Universal Robots URScript: MM_SIF408_Camera.script

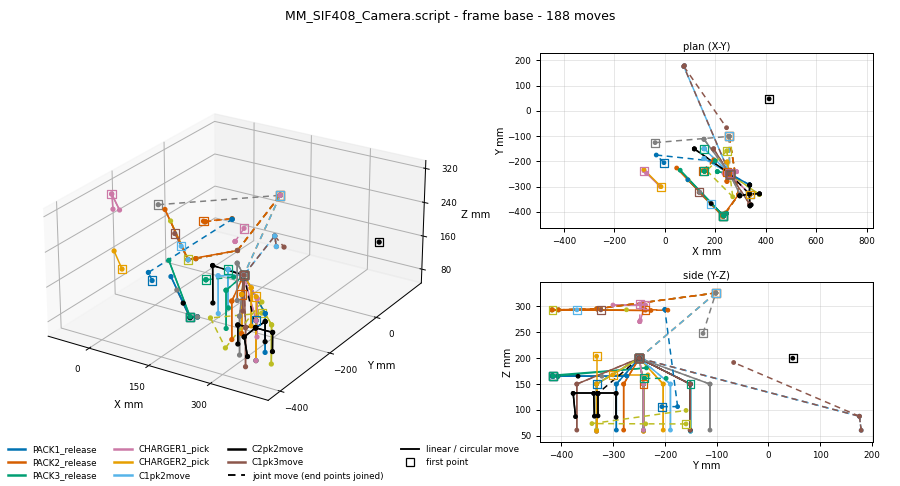
[picture p0: tool path of MM_SIF408_Camera.script in frame base, 188 of 288 moves have a stored position in this frame; points joined in program order, loops and branches not executed]
def MM_SIF408_Camera():
  global _hidden_verificationVariable=0
  step_count_84a8275e_68ac_46b0_8c6d_5b8d50443a58 = 0.0
  thread Step_Counter_Thread_a542c264_a21e_4968_aa71_40a8ac97ed48():
    while (True):
      step_count_84a8275e_68ac_46b0_8c6d_5b8d50443a58 = step_count_84a8275e_68ac_46b0_8c6d_5b8d50443a58 + 1.0
      sync()
    end
  end
  run Step_Counter_Thread_a542c264_a21e_4968_aa71_40a8ac97ed48()
  set_standard_analog_input_domain(0, 1)
  set_standard_analog_input_domain(1, 1)
  set_tool_analog_input_domain(0, 1)
  set_tool_analog_input_domain(1, 1)
  set_analog_outputdomain(0, 0)
  set_analog_outputdomain(1, 0)
  set_input_actions_to_default()
  modbus_add_signal("130.130.130.202", 255, 128, 2, "mm_insp_id", False)
  modbus_set_signal_update_frequency("mm_insp_id", 10)
  modbus_add_signal("130.130.130.202", 255, 129, 2, "mm_pht_stp_done", False)
  modbus_set_signal_update_frequency("mm_pht_stp_done", 10)
  modbus_add_signal("130.130.130.202", 255, 130, 2, "mm_res_ver", False)
  modbus_set_signal_update_frequency("mm_res_ver", 10)
  modbus_add_signal("130.130.130.202", 255, 131, 2, "c1_recorrect", False)
  modbus_set_signal_update_frequency("c1_recorrect", 10)
  modbus_add_signal("130.130.130.202", 255, 132, 2, "c2_recorrect", False)
  modbus_set_signal_update_frequency("c2_recorrect", 10)
  modbus_add_signal("130.130.130.202", 255, 133, 2, "c3_reconnect", False)
  modbus_set_signal_update_frequency("c3_reconnect", 10)
  modbus_add_signal("130.130.130.202", 255, 134, 2, "c4_reconnect", False)
  modbus_set_signal_update_frequency("c4_reconnect", 10)
  modbus_add_signal("130.130.130.202", 255, 135, 3, "mm_recv_inst", False)
  modbus_set_signal_update_frequency("mm_recv_inst", 10)
  modbus_add_signal("130.130.130.202", 255, 136, 3, "mm_pht_rdy_stp", False)
  modbus_set_signal_update_frequency("mm_pht_rdy_stp", 10)
  modbus_set_runstate_dependent_choice("mm_recv_inst",0)
  modbus_set_runstate_dependent_choice("mm_pht_rdy_stp",0)
  set_safety_mode_transition_hardness(1)
  set_tool_communication(True, 19200, 0, 1, 3.5, 3.5)
  set_tool_output_mode(1)
  set_tool_digital_output_mode(0, 1)
  set_tool_digital_output_mode(1, 1)
  set_tool_voltage(24)
  rtde_set_watchdog("speed_slider_mask", 10.0, "pause")
  rtde_set_watchdog("input_bit_registers0_to_31", 10.0, "pause")
  rtde_set_watchdog("input_bit_registers32_to_63", 10.0, "pause")
  set_tcp(p[0.0,0.0,0.105,0.0,0.0,0.0])
  set_gravity([0.0, 0.0, 9.82])
  set_target_payload(0.750000, [0.000000, 0.000000, 0.000000], [0.000000, 0.000000, 0.000000, 0.000000, 0.000000, 0.000000])
  global Plane_1_Pack=p[0.24802604835791223,-0.16109825037384065,0.07343232674968579,1.5770610514332666E-4,-1.6911666992609967E-4,-2.356123162082294]
  global Plane_2_Charger=p[-0.020825889928195812,-0.20923497632823723,0.10484675194267869,0.7321684888960871,-1.7600381110435173,-1.7743768301112888]
  global Plane_3_C1move=p[0.13168317783925995,-0.24026381339900515,0.1798744586307036,-1.7458660631601477,-0.7339675944130294,-1.7576520505834232]
  global abajo=p[0.236823956197105,-0.3085340218782548,0.07438383757948624,1.59760453662429E-5,-1.9018418942279844E-5,0.7930744342156013]
  global ChargerSafe_p=p[-.038219888098, -.126109356632, .247864627735, .768372410548, 1.381786852190, .427050797557]
  global ChargerSafe_q=[-2.290328532835165, -1.588600530279578, -1.8552938851973906, 3.426818033809969, -3.618186683716541, 5.475553405421589]
  global UL_HomePos_p=p[.254854540361, -.101396521086, .326005914920, .372294290291, 1.604272927406, .848817535244]
  global UL_HomePos_q=[-0.4437336060017767, -1.2677181226029575, -1.7403695179117786, 2.998681575604259, -2.3285643390928694, 5.484779635767351]
  global HomePos_p=p[.155172845975, -.134373233263, .327052937324, .372294290291, 1.604272927406, .848817535244]
  global HomePos_q=[-0.4437336060017767, -1.2677181226029575, -1.7403695179117786, 2.998681575604259, -2.3285643390928694, 5.484779635767351]
  global Waypoint_7_p=p[.235254426101, -.248279333010, .270600000000, -2.208471707321, 2.232557069129, -.003211421070]
  global Waypoint_7_q=[-0.4211163855529749, -1.695971462694982, -1.0919650932703284, 4.362995611362158, -4.714225695778342, 5.8733503607511075]
  global pl1_PK1up_2_p=p[.337707127627, -.331640151444, .150000000000, 2.209085410286, -2.230597199976, -.000628263705]
  global pl1_PK1up_2_q=[-0.4955539304835268, -2.270575736419687, -0.8287766003440309, 4.671022250611815, -4.717607275805612, 5.796412978798368]
  global pl1_PK1_1_p=p[.337708753286, -.331636321686, .059000000000, -2.208471682409, 2.232557092114, -.003211423953]
  global pl1_PK1_1_q=[-0.4967761842328837, -2.335801782331149, -1.1486863800200018, 5.0595087773604295, -4.714537561241828, 5.795733238729151]
  global pl1_PK1up_3_p=p[.337708753384, -.331636321739, .150000000045, -2.208471682402, 2.232557092122, -.003211423956]
  global pl1_PK1up_3_q=[-0.49668749848969007, -2.2676720609196863, -0.8351585073611147, 4.677851316512167, -4.714970187304847, 5.796430139558901]
  global Pack_aprox_1_p=p[.337708753236, -.331636321646, .203842313590, -2.208471707275, 2.232557069151, -.003211421080]
  global Pack_aprox_1_q=[-0.496372010829246, -2.3390319457501776, -0.44938640702618393, 4.363438999629054, -4.7153696447693765, 5.797111330864401]
  global pl1_PK2up_2_p=p[.246731843456, -.241011109916, .150000000097, 2.216981679034, -2.216426599865, .020673083567]
  global pl1_PK2up_2_q=[-0.3786656314116641, -1.6678189422546685, -1.7017298433113472, 4.951739825014103, -4.725262422761782, 5.9037751461208146]
  global p1_PK2_1_p=p[.246740908824, -.241008821032, .059000000000, 2.216983575726, -2.216446161785, .020720900301]
  global p1_PK2_1_q=[-0.3783922270214717, -1.8357706067986292, -1.9724640638814472, 5.390461636587837, -4.7249178522998685, 5.903567044989178]
  global pl1_PK2up_3_p=p[.246731843456, -.241011109916, .150000000097, 2.216981679034, -2.216426599865, .020673083567]
  global pl1_PK2up_3_q=[-0.3786656314116641, -1.6678189422546685, -1.7017298433113472, 4.951739825014103, -4.725262422761782, 5.9037751461208146]
  global Pack_aprox_3_p=p[.256529190168, -.247747736730, .304914735485, 2.216953502726, -2.216313122856, .021013179600]
  global Pack_aprox_3_q=[-0.45002005833990744, -1.7307120515452397, -1.4394096347220158, 4.751286312039589, -4.721256037152659, 5.839676484550372]
  global pl1_PK3up_2_p=p[.155982981866, -.150235111585, .149999999926, 2.204929412033, -2.228375225269, .020999038139]
  global pl1_PK3up_2_q=[-0.10405906347300053, -1.0147413698994976, -2.1858064021499084, 4.779384433270495, -4.726165068369075, 6.189377387251229]
  global pl1_PK3_1_p=p[.155974863337, -.150228231486, .059000001039, 2.204948002857, -2.228371305887, .020942580810]
  global pl1_PK3_1_q=[-0.10298431003644293, -1.1927496937335196, -2.5640957297909734, 5.335649879847573, -4.725692754745326, 6.190048722360077]
  global pl1_PK3up_3_p=p[.155982981866, -.150235111585, .149999999926, 2.204929412033, -2.228375225269, .020999038139]
  global pl1_PK3up_3_q=[-0.10405906347300053, -1.0147413698994976, -2.1858064021499084, 4.779384433270495, -4.726165068369075, 6.189377387251229]
  global C1_aprox1_p=p[-.133997460325, -.084557413006, .272269436052, .701218117570, 1.477825459734, .526200205067]
  global C1_aprox1_q=[-2.2378674310252507, -1.4936566577695842, -1.8069725022863468, 3.3775135356243458, -3.7069992982634132, 5.561485476738353]
  global C1_aprox2_p=p[-.161176845609, -.139586814883, .246569453044, 1.098520360937, 1.128202257975, .008787883398]
  global C1_aprox2_q=[-2.290389491672745, -1.5926356378882414, -1.8508182165530052, 3.416578818412902, -3.08727806453735, 5.46338959297019]
  global pl2_C1out_p=p[-.081795651010, -.237359145335, .302681515088, 1.127755706772, 1.089516743668, .021133838194]
  global pl2_C1out_q=[-2.1527147663452713, -1.5258578937050737, -1.651927109692683, 3.1816164398943436, -2.933001372406314, 5.5322042515010725]
  global pl2_C1_p=p[-.017768025182, -.300045052232, .302675455173, 1.127760213979, 1.089524808365, .021174235875]
  global pl2_C1_q=[-1.7215911662326384, -1.440872933618568, -1.7285842813986232, 3.1710747540129964, -2.5018731616546397, 5.52987656907406]
  global pl2_C1out_1_p=p[-.081795651010, -.237359145335, .302681515088, 1.127755706772, 1.089516743668, .021133838194]
  global pl2_C1out_1_q=[-2.1527147663452713, -1.5258578937050737, -1.651927109692683, 3.1816164398943436, -2.933001372406314, 5.5322042515010725]
  global pl2_C1scanner_p=p[-.072271028715, -.247338608301, .273275423406, 1.126803161894, 1.098257320894, .000808970523]
  global pl2_C1scanner_q=[-2.0835769100910424, -1.5156384620851568, -1.7953574861073918, 3.295232058172276, -2.8555002423783993, 5.496044985177414]
  global Pre_take_C2_p=p[-.157335508009, -.158680681186, .166974168240, 1.104025120675, 1.106172856258, .007095934659]
  global Pre_take_C2_q=[-2.170749334524068, -1.7352002992733144, -2.1267825877515776, 3.898556352135264, -2.960911303703792, 43.23650170495587]
  global Take_C2_p=p[-.014627410872, -.300575637934, .167809324670, 1.104025120587, 1.106172856207, .007095934493]
  global Take_C2_q=[-1.709235364834873, -1.6635052137678379, -2.2123391847121, 3.8869296419309585, -2.4994445138594434, 43.20973984887429]
  global Pre_take_C2_1_p=p[-.082686187568, -.232516861148, .167809324647, 1.104025120675, 1.106172856258, .007095934659]
  global Pre_take_C2_1_q=[-2.170749334524068, -1.7352002992733127, -2.1267825877515767, 3.898556352135266, -2.960911303703792, 43.23650170495587]
  global scanner_p=p[-.145597174960, -.172184123463, .273557709852, 1.126803161894, 1.098257320894, .000808970523]
  global scanner_q=[-2.0835769100910424, -1.5156384620851568, -1.7953574861073918, 3.295232058172276, -2.8555002423783993, 5.496044985177414]
  global C1mov_aprox_p=p[.308850778448, -.227461967730, .296313717128, 1.553122177506, .476375466750, -.700321395454]
  global C1mov_aprox_q=[-0.10623925922560318, -2.0247123961220943, -1.0679247316199865, 3.266489218161886, 0.052716603751015056, 5.361832612950986]
  global C1premove_2_p=p[.272288632653, -.321363961865, .303273960249, 1.719848172269, .285921327209, -.876957313116]
  global C1premove_2_q=[-0.3141074377311224, -1.9847352067666773, -1.152918690164526, 3.8692477100322447, 0.14198410920567195, 4.806071525474792]
  global pl3C1mov_ini_p=p[.182437129429, -.369644570295, .293330233139, 1.719847916544, .285941799097, -.876964145719]
  global pl3C1mov_ini_q=[-0.21453829232660748, -1.7685869829425869, -1.3791136381257303, 3.5854983324619933, 0.22740921363954233, 5.104717641505136]
  global pl3C1mback_p=p[.230951893202, -.418172131116, .293330097072, 1.719919114660, .285845055246, -.876955330681]
  global pl3C1mback_q=[-0.3165798667735258, -1.9909638241500476, -1.1468897455162494, 3.8811135011932274, 0.14018099976871434, 4.794327887884211]
  global pl3C1mback_apr_p=p[.240989471742, -.405297152942, .293331860507, 1.719848172156, .285921327154, -.876957313181]
  global pl3C1mback_apr_q=[-0.2753928168585782, -2.044774562435851, -1.0268096531551087, 3.653287708096954, 0.17311250712896362, 4.957879924004878]
  global UL_C1mov_aprox_p=p[.292891726775, -.331236745905, .295323683501, 1.553128130654, .476365407288, -.700325429374]
  global UL_C1mov_aprox_q=[-0.015735928212301076, -2.005986352960104, -1.0958646535873413, 3.2128893572041015, 0.13516616821289062, 5.424745559692383]
  global C2mov_aprox_p=p[.308833685463, -.227493882217, .174984383548, 1.553153487693, .476404540855, -.700571987051]
  global C2mov_aprox_q=[-0.107398811970846, -2.1403310934649866, -1.4719222227679651, 3.7666635513305664, 0.053114086389541626, 5.3811211585998535]
  global C2premove_2_p=p[.232175782362, -.415341220864, .165130240991, 1.745215389245, .199339967791, -1.099603067118]
  global C2premove_2_q=[-0.32663041750063115, -2.425627370873922, -0.9553382396697998, 3.6024443346210937, 0.29616692662239075, 5.22719669342041]
  global pl3C2mov_ini_p=p[.184286098126, -.367451536649, .165130240985, 1.745215389239, .199339967789, -1.099603067120]
  global pl3C2mov_ini_q=[-0.2396854698372417, -2.146879351703892, -1.4525406721582996, 3.7744590259789557, 0.38210751406196664, 5.2765130097251385]
  global pl3C2mback_p=p[.233731308910, -.416893857772, .165125834654, 1.745193719612, .199388652546, -1.099615399359]
  global pl3C2mback_q=[-0.32897164146040225, -2.4362316765895464, -0.9354621316722733, 3.594750230756894, 0.2938300334693391, 5.225506379883964]
  global pl3C2mback_apr_p=p[.244352223177, -.406272943615, .165125834657, 1.745193719588, .199388652550, -1.099615399369]
  global pl3C2mback_apr_q=[-0.2965665658105694, -2.4580305155795994, -0.8921927447881162, 3.551827498712303, 0.325544655967972, 5.248086636346506]
  global C1premove_3_p=p[.272288632653, -.321363961865, .303273960249, 1.719848172269, .285921327209, -.876957313116]
  global C1premove_3_q=[-0.3141074377311197, -1.9847352067666932, -1.1529186901644977, 3.869247710032223, 0.1419841092056745, 4.806071525474801]
  global pl3C1mov_ini_1_p=p[.136206182359, -.323413227205, .293329783718, 1.719843595479, .285997618514, -.877006764163]
  global pl3C1mov_ini_1_q=[-0.06361796225828531, -1.526354880356469, -1.619649605913061, 3.4154179150228465, 0.37045800628523196, 5.280448618100277]
  global pl3C1mback_1_p=p[.230951893193, -.418172131107, .293330097072, 1.719919114661, .285845055244, -.876955330680]
  global pl3C1mback_1_q=[-0.31657986675838057, -1.9909638241092953, -1.146889745557237, 3.881113501127934, 0.140180999780916, 4.794327887952139]
  global pl3C1mback_ap_1_p=p[.240989471377, -.405297153409, .293331860507, 1.719848172161, .285921327141, -.876957313189]
  global pl3C1mback_ap_1_q=[-0.2753928183421852, -2.044774560646961, -1.0268096569026657, 3.6532877147078273, 0.17311250588896365, 4.957879919281967]
  global pl3C2mov_ini_1_p=p[.138302268197, -.321469744604, .165129683929, 1.745209365041, .199365354932, -1.099621614261]
  global pl3C2mov_ini_1_q=[-0.11751452597140677, -1.9094658816367902, -1.8258869083293803, 3.8718451206663453, 0.5033504501004973, 5.319132560338594]
  global pl3C2mback_1_p=p[.233731306511, -.416893855378, .165125834660, 1.745193719657, .199388652393, -1.099615399351]
  global pl3C2mback_1_q=[-0.32897163787581807, -2.436231660170979, -0.935462162493657, 3.5947502426879394, 0.2938300370981234, 5.225506382567149]
  global pl3C2mback_ap_1_p=p[.244352222764, -.406272944029, .165125834657, 1.745193719588, .199388652550, -1.099615399369]
  global pl3C2mback_ap_1_q=[-0.2965665670586013, -2.4580305146957797, -0.892192746533599, 3.551827500318334, 0.3255446547441763, 5.248086635558534]
  global C1premove_4_p=p[.229536899103, -.416749725638, .293331860476, 1.719848172269, .285921327209, -.876957313116]
  global C1premove_4_q=[-0.3141074377311197, -1.9847352067666932, -1.1529186901644977, 3.869247710032223, 0.1419841092056745, 4.806071525474801]
  global pl3C1mov_ini_2_p=p[.092918330971, -.273904081257, .293515218460, 1.738538514888, .142309381755, -1.092432624406]
  global pl3C1mov_ini_2_q=[0.06853852740443775, -1.4945684218776059, -1.672527393380168, 3.253710061566366, 0.7126236314348806, 5.413101835930292]
  global pl3C1mback_2_p=p[.230951893193, -.418172131107, .293330097072, 1.719919114661, .285845055244, -.876955330680]
  global pl3C1mback_2_q=[-0.31657986675838057, -1.9909638241092953, -1.146889745557237, 3.881113501127934, 0.140180999780916, 4.794327887952139]
  global pl3C1mback_ap_2_p=p[.240989471377, -.405297153409, .293331860507, 1.719848172161, .285921327141, -.876957313189]
  global pl3C1mback_ap_2_q=[-0.2753928183421852, -2.044774560646961, -1.0268096569026657, 3.6532877147078273, 0.17311250588896365, 4.957879919281967]
  global pl3C2mov_ini_2_p=p[.091379813932, -.273144720278, .165459521490, 1.781697925685, .141363795277, -1.113411595331]
  global pl3C2mov_ini_2_q=[0.05406405031681061, -1.6675650082030238, -2.112321376800537, 3.9155165392109375, 0.7278146743774414, 5.354104042053223]
  global pl3C2mback_2_p=p[.233731306511, -.416893855378, .165125834660, 1.745193719657, .199388652393, -1.099615399351]
  global pl3C2mback_2_q=[-0.32897163787581807, -2.436231660170979, -0.935462162493657, 3.5947502426879394, 0.2938300370981234, 5.225506382567149]
  global pl3C2mback_ap_2_p=p[.244352222764, -.406272944029, .165125834657, 1.745193719588, .199388652550, -1.099615399369]
  global pl3C2mback_ap_2_q=[-0.2965665670586013, -2.4580305146957797, -0.892192746533599, 3.551827500318334, 0.3255446547441763, 5.248086635558534]
  global C1premove_5_p=p[.229536899103, -.416749725638, .293331860476, 1.719848172269, .285921327209, -.876957313116]
  global C1premove_5_q=[-0.3141074377311197, -1.9847352067666932, -1.1529186901644977, 3.869247710032223, 0.1419841092056745, 4.806071525474801]
  global pl3C1mov_ini_3_p=p[.047250403200, -.226621485350, .292173929776, 1.766368897888, .056774167404, -1.124179153332]
  global pl3C1mov_ini_3_q=[0.3235071206959865, -1.245212886825775, -1.8594057987392762, 3.185909029445348, 1.0430962588709336, 5.460546383776747]
  global pl3C1mback_3_p=p[.230951893193, -.418172131107, .293330097072, 1.719919114661, .285845055244, -.876955330680]
  global pl3C1mback_3_q=[-0.31657986675838057, -1.9909638241092953, -1.146889745557237, 3.881113501127934, 0.140180999780916, 4.794327887952139]
  global pl3C1mback_ap_3_p=p[.240989471377, -.405297153409, .293331860507, 1.719848172161, .285921327141, -.876957313189]
  global pl3C1mback_ap_3_q=[-0.2753928183421852, -2.044774560646961, -1.0268096569026657, 3.6532877147078273, 0.17311250588896365, 4.957879919281967]
  global pl3C2mov_ini_3_p=p[.061143010327, -.235334306883, .181227706054, 1.503856780720, 1.284559411089, -2.269349078019]
  global pl3C2mov_ini_3_q=[0.18262362480163574, -1.751157899896139, -2.196155071258545, 3.7787043291279296, 0.9670724868774414, 4.188342571258545]
  global pl3C2mback_3_p=p[.233733613016, -.416894540060, .167000000579, 1.745191210241, .199403215391, -1.099619453893]
  global pl3C2mback_3_q=[-0.32896921430330206, -2.434090063678788, -0.9304886701700523, 3.587597377758055, 0.2938370293056218, 5.225534676226004]
  global pl3C2mback_ap_3_p=p[.244352222764, -.406272944029, .165125834657, 1.745193719588, .199388652550, -1.099615399369]
  global pl3C2mback_ap_3_q=[-0.2965665670586013, -2.4580305146957797, -0.892192746533599, 3.551827500318334, 0.3255446547441763, 5.248086635558534]
  global UL_Pack_aprox_1_p=p[.257007851030, -.249235402177, .199905770770, 2.216850868158, -2.216446826465, .020822233207]
  global UL_Pack_aprox_1_q=[-0.45005588634680826, -1.730736453439805, -1.4394333534656631, 4.751226321242292, -4.7211960511095565, 5.839748112766433]
  global Belt_up_p=p[.413476933324, .047261308085, .199999999963, 2.199613607438, -2.234996179221, -.010379605365]
  global Belt_up_q=[0.4309097260458052, -1.9931567946711226, -1.0372145384205904, 4.595425950236857, -4.710855873196678, 6.729752451726602]
  global Belt_end_p=p[.019916769813, .441267430538, .304995973614, 2.199613607437, -2.234996179221, -.010379605365]
  global Belt_end_q=[1.8242716611485537, -2.118169382086794, -0.8490772289913693, 4.542803716350939, -4.707187498038789, 8.123017388538901]
  global Belt_down_p=p[-.071089290030, .533903585105, .161097633183, 2.199613607441, -2.234996179222, -.010379605363]
  global Belt_down_q=[1.947690189337532, -2.739873965415446, -0.3744445307036006, 4.690862938702149, -4.708236482539375, 8.244824259195594]
  global Pallet_prepick_p=p[.291447662150, -.062412426099, .254999999861, -3.141571401839, .001766180255, -.000038515322]
  global Pallet_prepick_q=[0.2422024256803905, -1.4673072639925095, -1.8978277566501056, 4.937857988785715, -4.7134268153705925, 4.955414063945926]
  global Pallet_pick_p=p[.291687034034, -.062651798319, .120335378275, -3.141571401871, .001766180260, -.000038515309]
  global Pallet_pick_q=[0.24172604282357715, -1.8270419989802704, -2.279616813584795, 5.6793807162253, -4.713012522321009, 4.954324153844183]
  global Pallet_release_p=p[.439378778235, -.217433323049, .234644516766, 2.229958612885, -2.203829311865, -.018817956446]
  global Pallet_release_q=[-0.18887788454164678, -2.374524255792135, -0.7392873764038086, 4.672313852901123, -4.706885520611898, 43.77889194485364]
  global D1_pallet_down_p=p[.442212069240, -.227560876465, .172521257618, 2.228035125756, -2.208520596470, -.014538793865]
  global D1_pallet_down_q=[-0.20933802990501782, -2.4453334804264983, -0.897326547308384, 4.905175531048007, -4.714222643234424, 6.063467806195847]
  global D1_pallet_up_p=p[.442218220834, -.227551384112, .188994489016, 2.228075464710, -2.208518983992, -.014530549009]
  global D1_pallet_up_q=[-0.20930559602697585, -2.430424251311435, -0.8470119229044197, 4.839971101978789, -4.714275805486577, 6.063594780073675]
  global D2_pallet_down_p=p[.404813401489, -.190162208820, .172521257584, 2.228035125755, -2.208520596469, -.014538793864]
  global D2_pallet_down_q=[-0.14314067688719945, -2.216033459875792, -1.3154267742044423, 5.0940825977907185, -4.71290441465381, 6.129949327460881]
  global D2_pallet_up_p=p[.404818650929, -.190154225512, .188994456919, 2.228042788212, -2.208499206561, -.014554532536]
  global D2_pallet_up_q=[-0.1431301070271589, -2.1913775737552568, -1.2753562616135667, 5.029342640058151, -4.712967534795309, 6.130053919158604]
  global D_UP_p=p[.422408824246, -.207743926117, .239494454368, 2.228032653101, -2.208505113638, -.014552037770]
  global D_UP_q=[-0.17597556501482003, -2.260678982325242, -0.9150656238765071, 4.738294750754857, -4.713841925756468, 6.097433375695097]
  global Pick_canister_p=p[.291446154867, -.062406995508, .164869940287, 3.141592162399, -.001756769940, -.000000000014]
  global Pick_canister_q=[0.24264195582142573, -1.6535789093299211, -2.191154567723123, 5.417426855963988, -4.713095863731711, 4.955409408171661]
  global Canister_aprox_p=p[.256979451068, -.249233253173, .199827674461, -3.136885319000, -.009569255568, -.021659245929]
  global Canister_aprox_q=[-0.4616465269995551, -1.7360003057116913, -1.4335725672291586, 4.750709769138723, -4.700207671443079, 4.251542634448455]
  global pl1Canister11up_p=p[.336350464321, -.369866932340, .150000000083, -3.136593313961, .019217351964, -.022201258143]
  global pl1Canister11up_q=[-0.5726090784291946, -2.4418729013936917, -0.5224593275151035, 4.546353320527715, -4.704289190477125, 4.151008395473293]
  global pl1Canister11_p=p[.336357723078, -.369867631038, .061145566587, -3.136612210135, .019157506079, -.022245010591]
  global pl1Canister11_q=[-0.572826076704029, -2.4569712728924884, -0.9138843149714617, 4.952901055542541, -4.703795635890442, 4.1501571565519075]
  global pl1Canist11up_1_p=p[.336350464321, -.369866932340, .150000000083, -3.136593313961, .019217351964, -.022201258143]
  global pl1Canist11up_1_q=[-0.5726090784291946, -2.4418729013936917, -0.5224593275151035, 4.546353320527715, -4.704289190477125, 4.151008395473293]
  global pl1Canister12up_p=p[.298153540198, -.331694754285, .150007342120, -3.136621792734, .019286306832, -.022194259920]
  global pl1Canister12up_q=[-0.5465683593869741, -2.120773045552329, -1.0831491423228998, 4.786258609062243, -4.703779014513574, 4.177393307867642]
  global pl1Canister12_p=p[.298143582441, -.331696625785, .061149999871, -3.136626162687, .019247363787, -.022096975362]
  global pl1Canister12_q=[-0.5465714266142632, -2.2160951455646867, -1.3565901714123374, 5.154963690976856, -4.7034223607341525, 4.176791699247043]
  global pl1Canist12up_p=p[.298153540198, -.331694754285, .150007342120, -3.136621792734, .019286306832, -.022194259920]
  global pl1Canist12up_q=[-0.5465683593869741, -2.120773045552329, -1.0831491423228998, 4.786258609062243, -4.703779014513574, 4.177393307867642]
  global pl1Canister13up_p=p[.374537816791, -.331687146531, .150015810981, -3.136619406175, .019237380757, -.022264711560]
  global pl1Canister13up_q=[-0.4643338658946581, -2.442316652748496, -0.5220563892552521, 4.547652881108839, -4.705373559610073, 4.259290250429998]
  global pl1Canister13_p=p[.374545985810, -.331682716721, .061149999829, -3.136629406775, .019236100383, -.022255516426]
  global pl1Canister13_q=[-0.46453771018321, -2.457467394630512, -0.91341757602585, 4.954155961506957, -4.704889900391203, 4.258489906537653]
  global pl1Canist13up_p=p[.374537816791, -.331687146531, .150015810981, -3.136619406175, .019237380757, -.022264711560]
  global pl1Canist13up_q=[-0.4643338658946581, -2.442316652748496, -0.5220563892552521, 4.547652881108839, -4.705373559610073, 4.259290250429998]
  global pl1Canister14up_p=p[.336330607795, -.293522363561, .150011107923, -3.136629546068, .019289158132, -.022228268939]
  global pl1Canister14up_q=[-0.4251966381166685, -2.1211846936538965, -1.0830073081795701, 4.787864663493958, -4.7050309418466805, 4.298760368347635]
  global pl1Canister14_p=p[.336335318148, -.293517632066, .061149999854, -3.136629420012, .019273179784, -.022245472568]
  global pl1Canister14_q=[-0.4251873257470198, -2.2166025110200733, -1.356313960708941, 5.156593386691696, -4.704634340081428, 4.298186717117115]
  global pl1Canist14up_p=p[.336330607795, -.293522363561, .150011107923, -3.136629546068, .019289158132, -.022228268939]
  global pl1Canist14up_q=[-0.4251966381166685, -2.1211846936538965, -1.0830073081795701, 4.787864663493958, -4.7050309418466805, 4.298760368347635]
  global pl1Canister21up_p=p[.246459943118, -.279378602173, .149999999952, -3.136626514608, .019263293631, -.022177721988]
  global pl1Canister21up_q=[-0.49614297788228434, -1.7934998252046963, -1.5527667546686992, 4.929161353929084, -4.703382206933557, 4.228095404239039]
  global pl1Canister21_p=p[.246467584560, -.279383190210, .061149999911, -3.136638006086, .019282961512, -.022229330059]
  global pl1Canister21_q=[-0.49597489598953715, -1.9390884468122707, -1.8110151777666665, 5.3330289877846315, -4.703033107422948, 4.227767205442929]
  global pl1Canist21up_p=p[.246459943118, -.279378602173, .149999999952, -3.136626514608, .019263293631, -.022177721988]
  global pl1Canist21up_q=[-0.49614297788228434, -1.7934998252046963, -1.5527667546686992, 4.929161353929084, -4.703382206933557, 4.228095404239039]
  global pl1Canister22up_p=p[.208272148212, -.241193205819, .150003306894, -3.136643464341, .019296830424, -.022184759817]
  global pl1Canister22up_q=[-0.4436125089540992, -1.5581126114684194, -1.8175582052629409, 4.9591368063594485, -4.703320005381344, 4.280797124281543]
  global pl1Canister22_p=p[.208256539951, -.241202746053, .061150000042, -3.136657866228, .019341417812, -.022105213985]
  global pl1Canister22_q=[-0.4433111614091301, -1.7333759996286693, -2.0945701042378477, 5.411370009013545, -4.703018008912175, 4.280676323703759]
  global pl1Canist22up_p=p[.208272148212, -.241193205819, .150003306894, -3.136643464341, .019296830424, -.022184759817]
  global pl1Canist22up_q=[-0.4436125089540992, -1.5581126114684194, -1.8175582052629409, 4.9591368063594485, -4.703320005381344, 4.280797124281543]
  global pl1Canister23up_p=p[.284643813774, -.241199172618, .150006827810, -3.136661669469, .019231161685, -.022197158457]
  global pl1Canister23up_q=[-0.3508109448056631, -1.7942732105823094, -1.55236981917687, 4.931034981758261, -4.705006456230956, 4.373398315826753]
  global pl1Canister23_p=p[.284641075935, -.241198976068, .061150000034, -3.136649443855, .019225557575, -.022194958134]
  global pl1Canister23_q=[-0.3506478307729868, -1.9399572158942284, -1.810417285135463, 5.334757422603368, -4.704650614587632, 4.3730494634905135]
  global pl1Canist23up_p=p[.284643813774, -.241199172618, .150006827810, -3.136661669469, .019231161685, -.022197158457]
  global pl1Canist23up_q=[-0.3508109448056631, -1.7942732105823094, -1.55236981917687, 4.931034981758261, -4.705006456230956, 4.373398315826753]
  global pl1Canister24up_p=p[.246464039414, -.203015456599, .150011978778, -3.136644549445, .019244693507, -.022228356803]
  global pl1Canister24up_q=[-0.2736913755395003, -1.5591109418897666, -1.8171965078368988, 4.961396122163025, -4.705287873823389, 4.450674247838194]
  global pl1Canister24_p=p[.246467129077, -.203021157891, .061150000022, -3.136658282344, .019225825659, -.022276808744]
  global pl1Canister24_q=[-0.27337373427271494, -1.734578322002145, -2.0939539681865114, 5.413652548784269, -4.704956950161413, 4.450530201543874]
  global pl1Canist24up_p=p[.246464039414, -.203015456599, .150011978778, -3.136644549445, .019244693507, -.022228356803]
  global pl1Canist24up_q=[-0.2736913755395003, -1.5591109418897666, -1.8171965078368988, 4.961396122163025, -4.705287873823389, 4.450674247838194]
  global pl1Canister31up_p=p[.155364412123, -.189041063320, .150000000055, -3.136613410815, .019187170854, -.022197501856]
  global pl1Canister31up_q=[-0.3288822226749639, -1.1913084004043553, -2.102666050530644, 4.878552350783232, -4.703762338847596, 4.3955534108780325]
  global pl1Canister31_p=p[.155365259666, -.189053355267, .061149999919, -3.136645463737, .019287624373, -.022238923899]
  global pl1Canister31_q=[-0.328183994381555, -1.3847188447923529, -2.4385375393266147, 5.40787170967147, -4.703404125570061, 4.395937890351204]
  global pl1Canist31up_p=p[.155364412123, -.189041063320, .150000000055, -3.136613410815, .019187170854, -.022197501856]
  global pl1Canist31up_q=[-0.3288822226749639, -1.1913084004043553, -2.102666050530644, 4.878552350783232, -4.703762338847596, 4.3955534108780325]
  global pl1Canister32up_p=p[.117189342257, -.150860696616, .150005524247, -3.136623911855, .019189122514, -.022267192899]
  global pl1Canister32up_q=[-0.1678628950221963, -0.8536149997293281, -2.2406222928462185, 4.6801624025778334, -4.705228340517797, 4.55653702092194]
  global pl1Canister32_p=p[.117192263169, -.150855348673, .061149999923, -3.136598206080, .019170383080, -.022307375324]
  global pl1Canister32_q=[-0.16639080818160856, -0.9710665445221593, -2.6389983983667658, 5.196017023247391, -4.704725571277725, 4.557555732949546]
  global pl1Canist32up_p=p[.117189342257, -.150860696616, .150005524247, -3.136623911855, .019189122514, -.022267192899]
  global pl1Canist32up_q=[-0.1678628950221963, -0.8536149997293281, -2.2406222928462185, 4.6801624025778334, -4.705228340517797, 4.55653702092194]
  global pl1Canister33up_p=p[.193541863889, -.150860898824, .149994660583, -3.136618612022, .019260692512, -.022180376209]
  global pl1Canister33up_q=[-0.10719113286580395, -1.1920971966227603, -2.1029227596135787, 4.881294099178955, -4.706607546622787, 4.617272694029578]
  global pl1Canister33_p=p[.193538509583, -.150869194572, .061149999964, -3.136650190596, .019300801291, -.022186633135]
  global pl1Canister33_q=[-0.10647299906098695, -1.3859760263706322, -2.4384751591134517, 5.410733442156981, -4.70625882088552, 4.617639478983933]
  global pl1Canist3up_p=p[.193541863889, -.150860898824, .149994660583, -3.136618612022, .019260692512, -.022180376209]
  global pl1Canist3up_q=[-0.10719113286580395, -1.1920971966227603, -2.1029227596135787, 4.881294099178955, -4.706607546622787, 4.617272694029578]
  global pl1Canister34up_p=p[.155358907509, -.112676989149, .149989110165, -3.136623170857, .019217437448, -.022152214821]
  global pl1Canister34up_q=[0.11631304007801273, -0.8547182818400598, -2.2409702806927463, 4.682989059213618, -4.7092137851604186, 4.84069864317922]
  global pl1Canister34_p=p[.155359171614, -.112668335527, .061149999983, -3.136599245518, .019157377320, -.022123678598]
  global pl1Canister34_q=[0.11780488689936364, -0.9731786715922697, -2.639002513991065, 5.199468350304402, -4.7087158380308365, 4.841712610308623]
  global pl1Canist34up_p=p[.155358907509, -.112676989149, .149989110165, -3.136623170857, .019217437448, -.022152214821]
  global pl1Canist34up_q=[0.11631304007801273, -0.8547182818400598, -2.2409702806927463, 4.682989059213618, -4.7092137851604186, 4.84069864317922]
  global PL1orig_p=p[.246026678330, -.158971282208, .073007228186, 2.219356651567, -2.215959744177, .001661932884]
  global PL1orig_q=[-0.18321848717445732, -1.650301515916512, -2.1719116841803405, 5.390808490613271, -4.715603921456922, 43.806772121545094]
  global PL1_Xinc_p=p[.166244623352, -.236876442176, .073218191722, -2.227707236567, 2.207279081029, -.013912689784]
  global PL1_Xinc_q=[-0.5693064142400859, -1.6319163939130323, -2.197266413198509, 5.409843113333984, -4.707061464588999, 43.41306613297339]
  global PL1_Yinc_p=p[.269355357778, -.340629062826, .073711855978, -2.227717579915, 2.207348833273, -.013876628563]
  global PL1_Yinc_q=[-0.6463977997140873, -2.1810136419685904, -1.4014857458483148, 5.162812338981528, -4.709242148115926, 43.33404425900006]
  global PL1orig_aprox_p=p[.246033981666, -.158957981768, .099155627949, 2.219458391875, -2.215838784996, .001609603470]
  global PL1orig_aprox_q=[-0.18314598337275356, -1.5780762702689124, -2.099462273954118, 5.24610369379295, -4.714840127795956, 43.80628621235597]
  global PL2orig_p=p[-.003229150917, -.205640399391, .106466423235, 1.111938642798, 1.116313019605, -.009318675577]
  global PL2orig_q=[-1.8322987342458887, -1.7037047464663537, -2.6603252884447146, 4.35382993802417, -2.603727893625141, 43.18000988330823]
  global PL2orig_aprox_p=p[-.033671544119, -.175161726036, .106449683899, 1.112090219175, 1.116254642254, -.009214547123]
  global PL2orig_aprox_q=[-2.1803260742267003, -1.7785545498580575, -2.5452660819192814, 4.2936225942953055, -2.9518125548708642, 43.159379042433]
  global PL2_Xinc_p=p[.197521951224, -.199883729817, .294025184634, 1.711314537904, -.001132274929, -1.214674067413]
  global PL2_Xinc_q=[0.1331487908153166, -2.01646279427215, -1.0887761240875165, 3.1049269395316945, 0.9284476273978068, 43.19428862495026]
  global PL2_Yinc_p=p[.197511929610, -.199891220330, .294025466236, 1.711291012982, -.001165018329, -1.214712349834]
  global PL2_Yinc_q=[0.13311281774361472, -2.016462738750292, -1.0888000277574648, 3.104915080397602, 0.9284476596790521, 43.194312374048444]
  global PL3orig_p=p[.150709990552, -.237217505719, .292701269272, 1.711323215576, -.000932940983, -1.214583619475]
  global PL3orig_q=[0.021024057292553522, -1.852386997169262, -1.3261440483925107, 3.1791602623926636, 0.8167970371630613, 43.19285294310873]
  global PL3orig_aprox_p=p[.193869330701, -.194020123741, .292694213990, 1.711305461977, -.001081911433, -1.214588775499]
  global PL3orig_aprox_q=[0.1531582749196403, -1.9931843756183802, -1.1295440593242745, 3.1225419728801214, 0.9485012099752641, 43.19412039175612]
  global PL3_Yinc_p=p[.157174178700, -.239892124051, .293991340433, 1.711399733516, -.001116861407, -1.214495617214]
  global PL3_Yinc_q=[0.011247641968507693, -1.88431781885624, -1.277288508339872, 3.1621738720517953, 0.8069733867461313, 43.19318182229017]
  global PL3_Zinc_p=p[.157170549146, -.239892398942, .293996188669, 1.711450832864, -.001169657090, -1.214461082348]
  global PL3_Zinc_q=[0.011235663125033213, -1.8842940652136217, -1.2772527096703712, 3.1621858003444903, 0.8069853062504917, 43.193169935522164]
  global PL4orig_p=p[.157158684992, -.239339801716, .161007644274, 1.711387491122, -.001210651046, -1.214451224812]
  global PL4orig_q=[0.01215216802982777, -2.0520964439513243, -1.694253499649209, 3.7454203433719564, 0.8096201134725325, 43.19542486771209]
  global PL4_Yinc_p=p[.157163256893, -.239330967714, .161011336051, 1.711422577655, -.001236030276, -1.214391242535]
  global PL4_Yinc_q=[0.012188136314109421, -2.052048285439742, -1.6942654989969252, 3.74544440234104, 0.8096441220331281, 43.19542466043286]
  global PL4_Zinc_p=p[.157156911865, -.239332910309, .161012473804, 1.711414459593, -.001211752530, -1.214437913048]
  global PL4_Zinc_q=[0.012176151493264342, -2.052048250198637, -1.6942774518112742, 3.7454325182092822, 0.8096441571014674, 43.19540076045646]
  global pl4orig_aprox_p=p[.199450082365, -.197395229496, .161076818111, 1.711398106421, -.001038854369, -1.214385145570]
  global pl4orig_aprox_q=[0.1390013332442841, -2.1606690262247232, -1.5099980169371943, 3.669623723688836, 0.9357287798063281, 43.195794324527235]
  global Waypoint_4_p=p[.256544943431, -.247742607224, .304863195657, .008284518875, 3.136854174315, -.022033037887]
  global Waypoint_4_q=[-0.38625651994807697, -1.8351708851255397, -0.7419311404229436, 4.159360094661417, -4.7263968626605894, 1.1904072443380844]
  global Waypoint_1_p=p[.235234595082, -.248301819732, .270601973694, .024992169454, 3.127506406652, .007596517975]
  global Waypoint_1_q=[-0.4272355252220841, -1.6910316158263115, -1.101333190923703, 4.375854076692655, -4.70453828311887, 7.443212315149811]
  global Waypoint_6_p=p[.235234595082, -.248301819732, .270601973694, -2.222522309033, 2.201569466030, -.010351189186]
  global Waypoint_6_q=[-0.4272355607813232, -1.6910315116186894, -1.1013333658388174, 4.375854273122178, -4.704538225940382, 5.846962038903081]
  global Waypoint_8_p=p[.235234595082, -.248301819732, .270601973694, -3.136316875124, .041167434529, -.021881545292]
  global Waypoint_8_q=[-0.42723555732179364, -1.6910314987181305, -1.1013333854417962, 4.375854290982936, -4.704538231514219, 4.311888381664771]
  global Waypoint_3_p=p[.337708753264, -.331636321663, .059000000066, -2.208471683428, 2.232557091087, -.003211423699]
  global Waypoint_3_q=[-0.4967761842389473, -2.3358017822143826, -1.1486863798424043, 5.0595087769148, -4.714537561180646, 5.795733237802837]
  global Waypoint_2_p=p[.337708753384, -.331636321739, .150000000045, -2.208471682402, 2.232557092122, -.003211423956]
  global Waypoint_2_q=[-0.49668749848969007, -2.2676720609196863, -0.8351585073611147, 4.677851316512167, -4.714970187304847, 5.796430139558901]
  global abv_poke_p=p[.075553659734, .175874014996, .087825256700, 3.108109649460, -.004306961101, -.034888188980]
  global abv_poke_q=[1.8731590704078123, -0.971181369058062, -2.4874348601851306, 5.006233874433412, -4.680643336687123, 6.587372124760976]
  global poke_holder_p=p[.077973932283, .179375534722, .060695955510, -3.111112262565, .024392477457, .001431253159]
  global poke_holder_q=[1.9056804681185258, -0.9796989608329163, -2.646376911093853, 5.227700960448129, -4.7211359032678075, 6.632877911258849]
  global abv_p1_p=p[.334935679930, -.329214111758, .131999999184, -2.109648905195, 2.323247852764, .009014645382]
  global abv_p1_q=[-0.4969284969276311, -2.2563533146326664, -0.9365864808642748, 4.761336427125869, -4.7103366891602585, 5.881549525676308]
  global c1_approx_p=p[.337374582537, -.376881990518, .131999999304, -2.109648910489, 2.323247848134, .009014661822]
  global c1_approx_q=[-0.5806979591009238, -2.4896403156274416, -0.5112999914243233, 4.568923806038075, -4.71126690664721, 5.797560477468719]
  global c1_push_p=p[.342695385652, -.372415668050, .087155508836, -2.107961506896, 2.307043993240, .043173007855]
  global c1_push_q=[-0.5744441191302698, -2.509622713128561, -0.6771805882453918, 4.736850501015343, -4.693113748227255, 5.7971673011779785]
  global c2_approx_p=p[.297286965922, -.337154107499, .132000000000, -2.141999548083, 2.289060645038, -.067785858900]
  global c2_approx_q=[-0.5506265896671501, -2.1141620835550086, -1.1930945244392888, 4.923218214382089, -4.720816618378958, 5.797765699542333]
  global c2_push_p=p[.296718583911, -.335969607030, .087955366627, -2.117565997456, 2.284761326805, -.029540497124]
  global c2_push_q=[-0.5609849135028284, -2.1753393612303675, -1.2982627153396606, 5.071412372380056, -4.694436017666952, 5.7971673011779785]
  global c3_approx_p=p[.375393638462, -.328902332030, .131999999914, -2.141987159495, 2.289046676690, -.067761269924]
  global c3_approx_q=[-0.4501288764800222, -2.3700003994241325, -0.7546091883096189, 4.739777363135948, -4.725764373432657, 5.897879951222097]
  global c3_push_p=p[.375389246017, -.328911064812, .088566987758, -2.141999548079, 2.289060645035, -.067785858997]
  global c3_push_q=[-0.45021891619817467, -2.3888423492270476, -0.9248158427194433, 4.928837400788129, -4.7255485422144385, 5.897506011114244]
  global c4_approx_p=p[.336555809783, -.293980888045, .132000000000, -2.141999548075, 2.289060645038, -.067785859028]
  global c4_approx_q=[-0.41600961056622054, -2.1016052918357673, -1.2126420880461453, 4.929052171419869, -4.726534306791507, 5.9322718248887725]
  global c4_push_p=p[.336555809692, -.293980888005, .086064045175, -2.141999548076, 2.289060645037, -.067785859029]
  global c4_push_q=[-0.41600174030198467, -2.1539398343746736, -1.3513076433212667, 5.120055452553088, -4.726326233860483, 5.931993263961527]
  global Waypoint_5_p=p[.244816361443, -.066954461326, .191685498275, 2.579837129660, -1.535028578172, .328880261476]
  global Waypoint_5_q=[0.5165866017341614, -1.0633739990046998, -1.9963605403900146, 4.6344215112873535, -4.962536994610922, 6.3017221114235085]
  def PACK1_release():
    $ 223 "PACK1_release" "noBreak"
    $ 224 "MoveJ"
    $ 225 "HomePos" "breakAfter"
    movej(get_inverse_kin(pose_trans(HomePos_p, get_tcp_offset()), qnear=HomePos_q), a=1.3962634015954636, v=1.0471975511965976)
    $ 226 "Waypoint_7" "breakAfter"
    movej(get_inverse_kin(pose_trans(Waypoint_7_p, get_tcp_offset()), qnear=Waypoint_7_q), a=1.3962634015954636, v=1.0471975511965976)
    $ 227 "MoveL"
    $ 228 "pl1_PK1up_2" "breakAfter"
    movel(pose_trans(Plane_1_Pack, pose_trans(p[.061451264231, -.289311417922, -.073379282729, -.000157706105, .000169116670, 2.356123162082], pl1_PK1up_2_p)), a=1.2, v=0.25)
    $ 229 "MoveL"
    $ 230 "pl1_PK1_1" "breakAfter"
    movel(pose_trans(Plane_1_Pack, pose_trans(p[.061451264231, -.289311417922, -.073379282729, -.000157706105, .000169116670, 2.356123162082], pl1_PK1_1_p)), a=1.2, v=0.25)
    $ 231 "Set OuTNET_Gripper=0"
    write_output_integer_register(0, 0)
    $ 232 "Set OutNet_Tool=On"
    write_output_boolean_register(2, True)
    $ 233 "Wait: 2.0"
    sleep(2.0)
    $ 234 "Wait: 5.0"
    sleep(5.0)
    $ 235 "Set OutNet_Tool=On"
    write_output_boolean_register(2, True)
    $ 236 "Wait: 2.0"
    sleep(2.0)
    $ 237 "pl1_PK1up_3" "breakAfter"
    movel(pose_trans(Plane_1_Pack, pose_trans(p[.061451264231, -.289311417922, -.073379282729, -.000157706105, .000169116670, 2.356123162082], pl1_PK1up_3_p)), a=1.2, v=0.25)
    $ 238 "MoveJ"
    $ 239 "Pack_aprox_1" "breakAfter"
    movej(get_inverse_kin(pose_trans(Pack_aprox_1_p, get_tcp_offset()), qnear=Pack_aprox_1_q), a=1.3962634015954636, v=1.0471975511965976)
    $ 240 "HomePos" "breakAfter"
    movej(get_inverse_kin(pose_trans(HomePos_p, get_tcp_offset()), qnear=HomePos_q), a=1.3962634015954636, v=1.0471975511965976)
    $ 241 "Set OutNet_Tool=Off"
    write_output_boolean_register(2, False)
  end
  def PACK2_release():
    $ 242 "PACK2_release" "noBreak"
    $ 243 "MoveJ"
    $ 244 "HomePos" "breakAfter"
    movej(get_inverse_kin(pose_trans(HomePos_p, get_tcp_offset()), qnear=HomePos_q), a=1.3962634015954636, v=1.0471975511965976)
    $ 245 "Waypoint_7" "breakAfter"
    movej(get_inverse_kin(pose_trans(Waypoint_7_p, get_tcp_offset()), qnear=Waypoint_7_q), a=1.3962634015954636, v=1.0471975511965976)
    $ 246 "MoveL"
    $ 247 "pl1_PK2up_2" "breakAfter"
    movel(pose_trans(Plane_1_Pack, pose_trans(p[.061451264231, -.289311417922, -.073379282729, -.000157706105, .000169116670, 2.356123162082], pl1_PK2up_2_p)), a=1.2, v=0.25)
    $ 248 "MoveL"
    $ 249 "p1_PK2_1" "breakAfter"
    movel(pose_trans(Plane_1_Pack, pose_trans(p[.061451264231, -.289311417922, -.073379282729, -.000157706105, .000169116670, 2.356123162082], p1_PK2_1_p)), a=1.2, v=0.25)
    $ 250 "Set OuTNET_Gripper=0"
    write_output_integer_register(0, 0)
    $ 251 "Set OutNet_Tool=On"
    write_output_boolean_register(2, True)
    $ 252 "Wait: 2.0"
    sleep(2.0)
    $ 253 "Wait: 5.0"
    sleep(5.0)
    $ 254 "Set OutNet_Tool=On"
    write_output_boolean_register(2, True)
    $ 255 "Wait: 2.0"
    sleep(2.0)
    $ 256 "pl1_PK2up_3" "breakAfter"
    movel(pose_trans(Plane_1_Pack, pose_trans(p[.061451264231, -.289311417922, -.073379282729, -.000157706105, .000169116670, 2.356123162082], pl1_PK2up_3_p)), a=1.2, v=0.25)
    $ 257 "MoveJ"
    $ 258 "Pack_aprox_3" "breakAfter"
    movej(get_inverse_kin(pose_trans(Pack_aprox_3_p, get_tcp_offset()), qnear=Pack_aprox_3_q), a=1.3962634015954636, v=1.0471975511965976)
    $ 259 "HomePos" "breakAfter"
    movej(get_inverse_kin(pose_trans(HomePos_p, get_tcp_offset()), qnear=HomePos_q), a=1.3962634015954636, v=1.0471975511965976)
    $ 260 "Set OutNet_Tool=Off"
    write_output_boolean_register(2, False)
  end
  def PACK3_release():
    $ 261 "PACK3_release" "noBreak"
    $ 262 "MoveJ"
    $ 263 "HomePos" "breakAfter"
    movej(get_inverse_kin(pose_trans(HomePos_p, get_tcp_offset()), qnear=HomePos_q), a=1.3962634015954636, v=1.0471975511965976)
    $ 264 "Waypoint_7" "breakAfter"
    movej(get_inverse_kin(pose_trans(Waypoint_7_p, get_tcp_offset()), qnear=Waypoint_7_q), a=1.3962634015954636, v=1.0471975511965976)
    $ 265 "MoveL"
    $ 266 "pl1_PK3up_2" "breakAfter"
    movel(pose_trans(Plane_1_Pack, pose_trans(p[.061451264231, -.289311417922, -.073379282729, -.000157706105, .000169116670, 2.356123162082], pl1_PK3up_2_p)), a=1.2, v=0.25)
    $ 267 "MoveL"
    $ 268 "pl1_PK3_1" "breakAfter"
    movel(pose_trans(Plane_1_Pack, pose_trans(p[.061451264231, -.289311417922, -.073379282729, -.000157706105, .000169116670, 2.356123162082], pl1_PK3_1_p)), a=1.2, v=0.25)
    $ 269 "Set OuTNET_Gripper=0"
    write_output_integer_register(0, 0)
    $ 270 "Set OutNet_Tool=On"
    write_output_boolean_register(2, True)
    $ 271 "Wait: 2.0"
    sleep(2.0)
    $ 272 "Wait: 5.0"
    sleep(5.0)
    $ 273 "Set OutNet_Tool=On"
    write_output_boolean_register(2, True)
    $ 274 "Wait: 2.0"
    sleep(2.0)
    $ 275 "pl1_PK3up_3" "breakAfter"
    movel(pose_trans(Plane_1_Pack, pose_trans(p[.061451264231, -.289311417922, -.073379282729, -.000157706105, .000169116670, 2.356123162082], pl1_PK3up_3_p)), a=1.2, v=0.25)
    $ 276 "MoveJ"
    $ 277 "Pack_aprox_3" "breakAfter"
    movej(get_inverse_kin(pose_trans(Pack_aprox_3_p, get_tcp_offset()), qnear=Pack_aprox_3_q), a=1.3962634015954636, v=1.0471975511965976)
    $ 278 "HomePos" "breakAfter"
    movej(get_inverse_kin(pose_trans(HomePos_p, get_tcp_offset()), qnear=HomePos_q), a=1.3962634015954636, v=1.0471975511965976, r=0.005)
    $ 279 "Set OutNet_Tool=Off"
    write_output_boolean_register(2, False)
  end
  def CHARGER1_pick():
    $ 280 "CHARGER1_pick" "noBreak"
    $ 281 "MoveJ"
    $ 282 "HomePos" "breakAfter"
    movej(get_inverse_kin(pose_trans(HomePos_p, get_tcp_offset()), qnear=HomePos_q), a=1.3962634015954636, v=1.0471975511965976)
    $ 283 "Set OutNET_Done=Off"
    write_output_boolean_register(1, False)
    $ 284 "Set OutNet_Tool=Off"
    write_output_boolean_register(2, False)
    $ 285 "C1_aprox1" "breakAfter"
    movej(get_inverse_kin(pose_trans(C1_aprox1_p, get_tcp_offset()), qnear=C1_aprox1_q), a=1.3962634015954636, v=1.0471975511965976)
    $ 286 "C1_aprox2" "breakAfter"
    movej(get_inverse_kin(pose_trans(C1_aprox2_p, get_tcp_offset()), qnear=C1_aprox2_q), a=1.3962634015954636, v=1.0471975511965976)
    $ 287 "MoveL"
    $ 288 "pl2_C1out" "breakAfter"
    movel(pose_trans(Plane_2_Charger, pose_trans(p[-.160637607656, -.107017785098, .133972337005, -.732168488896, 1.760038111044, 1.774376830111], pl2_C1out_p)), a=1.2, v=0.25)
    $ 289 "MoveL"
    $ 290 "pl2_C1" "breakAfter"
    movel(pose_trans(Plane_2_Charger, pose_trans(p[-.160637607656, -.107017785098, .133972337005, -.732168488896, 1.760038111044, 1.774376830111], pl2_C1_p)), a=1.2, v=0.2)
    $ 291 "Set OuTNET_Gripper=5"
    write_output_integer_register(0, 5)
    $ 292 "Set OutNet_Tool=On"
    write_output_boolean_register(2, True)
    $ 293 "Wait: 2.0"
    sleep(2.0)
    $ 294 "Wait InNET_InPos=HI"
    while (read_input_boolean_register(1) == False):
      sync()
    end
    $ 295 "Set OutNet_Tool=Off"
    write_output_boolean_register(2, False)
    $ 296 "MoveL"
    $ 297 "pl2_C1out_1" "breakAfter"
    movel(pose_trans(Plane_2_Charger, pose_trans(p[-.160637607656, -.107017785098, .133972337005, -.732168488896, 1.760038111044, 1.774376830111], pl2_C1out_1_p)), a=1.2, v=0.2)
    $ 298 "MoveL"
    $ 299 "pl2_C1scanner" "breakAfter"
    movel(pose_trans(Plane_2_Charger, pose_trans(p[-.160637607656, -.107017785098, .133972337005, -.732168488896, 1.760038111044, 1.774376830111], pl2_C1scanner_p)), a=1.2, v=0.25)
    $ 300 "Wait: 2.0"
    sleep(2.0)
    $ 301 "C1_aprox2" "breakAfter"
    movej(get_inverse_kin(pose_trans(C1_aprox2_p, get_tcp_offset()), qnear=C1_aprox2_q), a=1.3962634015954636, v=1.0471975511965976)
    $ 302 "C1_aprox1" "breakAfter"
    movej(get_inverse_kin(pose_trans(C1_aprox1_p, get_tcp_offset()), qnear=C1_aprox1_q), a=1.3962634015954636, v=1.0471975511965976)
    $ 303 "HomePos" "breakAfter"
    movej(get_inverse_kin(pose_trans(HomePos_p, get_tcp_offset()), qnear=HomePos_q), a=1.3962634015954636, v=1.0471975511965976)
  end
  def CHARGER2_pick():
    $ 304 "CHARGER2_pick" "noBreak"
    $ 305 "MoveJ"
    $ 306 "HomePos" "breakAfter"
    movej(get_inverse_kin(pose_trans(HomePos_p, get_tcp_offset()), qnear=HomePos_q), a=1.3962634015954636, v=1.0471975511965976)
    $ 307 "C1_aprox1" "breakAfter"
    movej(get_inverse_kin(pose_trans(C1_aprox1_p, get_tcp_offset()), qnear=C1_aprox1_q), a=1.3962634015954636, v=1.0471975511965976)
    $ 308 "Pre_take_C2" "breakAfter"
    movej(get_inverse_kin(pose_trans(Pre_take_C2_p, get_tcp_offset()), qnear=Pre_take_C2_q), a=1.3962634015954636, v=1.0471975511965976)
    $ 309 "MoveL"
    $ 310 "Take_C2" "breakAfter"
    movel(pose_trans(Plane_2_Charger, pose_trans(p[-.160637607656, -.107017785098, .133972337005, -.732168488896, 1.760038111044, 1.774376830111], Take_C2_p)), a=1.2, v=0.2)
    $ 311 "Set OuTNET_Gripper=5"
    write_output_integer_register(0, 5)
    $ 312 "Set OutNet_Tool=On"
    write_output_boolean_register(2, True)
    $ 313 "Wait: 2.0"
    sleep(2.0)
    $ 314 "Wait InNET_InPos=HI"
    while (read_input_boolean_register(1) == False):
      sync()
    end
    $ 315 "Set OutNet_Tool=Off"
    write_output_boolean_register(2, False)
    $ 316 "MoveL"
    $ 317 "Pre_take_C2_1" "breakAfter"
    movel(pose_trans(Plane_2_Charger, pose_trans(p[-.160637607656, -.107017785098, .133972337005, -.732168488896, 1.760038111044, 1.774376830111], Pre_take_C2_1_p)), a=1.2, v=0.2)
    $ 318 "scanner" "breakAfter"
    movej(get_inverse_kin(pose_trans(scanner_p, get_tcp_offset()), qnear=scanner_q), a=1.3962634015954636, v=1.0471975511965976)
    $ 319 "C1_aprox1" "breakAfter"
    movej(get_inverse_kin(pose_trans(C1_aprox1_p, get_tcp_offset()), qnear=C1_aprox1_q), a=1.3962634015954636, v=1.0471975511965976)
    $ 320 "HomePos" "breakAfter"
    movej(get_inverse_kin(pose_trans(HomePos_p, get_tcp_offset()), qnear=HomePos_q), a=1.3962634015954636, v=1.0471975511965976)
  end
  def C1pk2move():
    $ 321 "C1pk2move" "noBreak"
    $ 322 "MoveJ"
    $ 323 "HomePos" "breakAfter"
    movej(get_inverse_kin(pose_trans(HomePos_p, get_tcp_offset()), qnear=HomePos_q), a=1.3962634015954636, v=1.0471975511965976)
    $ 324 "C1mov_aprox" "breakAfter"
    movej(get_inverse_kin(pose_trans(C1mov_aprox_p, get_tcp_offset()), qnear=C1mov_aprox_q), a=1.3962634015954636, v=1.0471975511965976)
    $ 325 "MoveL"
    $ 326 "C1premove_2" "breakAfter"
    movel(pose_trans(pose_trans(Plane_3_C1move, pose_trans(p[-.180543022068, -.262061738902, .078420930934, 1.745866063160, .733967594413, 1.757652050583], C1premove_2_p)), get_tcp_offset()), a=0.6, v=0.08)
    $ 327 "MoveL"
    $ 328 "pl3C1mov_ini" "breakAfter"
    movel(pose_trans(Plane_3_C1move, pose_trans(p[-.180543022068, -.262061738902, .078420930934, 1.745866063160, .733967594413, 1.757652050583], pl3C1mov_ini_p)), a=0.6, v=0.08)
    $ 329 "Wait: 1.0"
    sleep(1.0)
    $ 330 "pl3C1mback" "breakAfter"
    movel(pose_trans(Plane_3_C1move, pose_trans(p[-.180543022068, -.262061738902, .078420930934, 1.745866063160, .733967594413, 1.757652050583], pl3C1mback_p)), a=0.6, v=0.08)
    $ 331 "pl3C1mback_apr" "breakAfter"
    movel(pose_trans(Plane_3_C1move, pose_trans(p[-.180543022068, -.262061738902, .078420930934, 1.745866063160, .733967594413, 1.757652050583], pl3C1mback_apr_p)), a=0.6, v=0.08)
    $ 332 "MoveJ"
    $ 333 "UL_C1mov_aprox" "breakAfter"
    movej(get_inverse_kin(UL_C1mov_aprox_p, qnear=UL_C1mov_aprox_q), a=1.3962634015954636, v=1.0471975511965976)
    $ 334 "UL_HomePos" "breakAfter"
    movej(get_inverse_kin(UL_HomePos_p, qnear=UL_HomePos_q), a=1.3962634015954636, v=1.0471975511965976)
  end
  def C2pk2move():
    $ 335 "C2pk2move" "noBreak"
    $ 336 "MoveJ"
    $ 337 "HomePos" "breakAfter"
    movej(get_inverse_kin(pose_trans(HomePos_p, get_tcp_offset()), qnear=HomePos_q), a=1.3962634015954636, v=1.0471975511965976)
    $ 338 "C2mov_aprox" "breakAfter"
    movej(get_inverse_kin(pose_trans(C2mov_aprox_p, get_tcp_offset()), qnear=C2mov_aprox_q), a=1.3962634015954636, v=1.0471975511965976)
    $ 339 "MoveL"
    $ 340 "C2premove_2" "breakAfter"
    movel(pose_trans(Plane_3_C1move, pose_trans(p[-.180543022068, -.262061738902, .078420930934, 1.745866063160, .733967594413, 1.757652050583], C2premove_2_p)), a=0.6, v=0.08)
    $ 341 "MoveL"
    $ 342 "pl3C2mov_ini" "breakAfter"
    movel(pose_trans(Plane_3_C1move, pose_trans(p[-.180543022068, -.262061738902, .078420930934, 1.745866063160, .733967594413, 1.757652050583], pl3C2mov_ini_p)), a=0.6, v=0.08)
    $ 343 "Wait: 1.0"
    sleep(1.0)
    $ 344 "pl3C2mback" "breakAfter"
    movel(pose_trans(Plane_3_C1move, pose_trans(p[-.180543022068, -.262061738902, .078420930934, 1.745866063160, .733967594413, 1.757652050583], pl3C2mback_p)), a=0.6, v=0.08)
    $ 345 "pl3C2mback_apr" "breakAfter"
    movel(pose_trans(Plane_3_C1move, pose_trans(p[-.180543022068, -.262061738902, .078420930934, 1.745866063160, .733967594413, 1.757652050583], pl3C2mback_apr_p)), a=0.6, v=0.08)
    $ 346 "MoveJ"
    $ 347 "C2mov_aprox" "breakAfter"
    movej(get_inverse_kin(pose_trans(C2mov_aprox_p, get_tcp_offset()), qnear=C2mov_aprox_q), a=1.3962634015954636, v=1.0471975511965976)
    $ 348 "HomePos" "breakAfter"
    movej(get_inverse_kin(pose_trans(HomePos_p, get_tcp_offset()), qnear=HomePos_q), a=1.3962634015954636, v=1.0471975511965976)
  end
  def C1pk3move():
    $ 349 "C1pk3move" "noBreak"
    $ 350 "MoveJ"
    $ 351 "HomePos" "breakAfter"
    movej(get_inverse_kin(pose_trans(HomePos_p, get_tcp_offset()), qnear=HomePos_q), a=1.3962634015954636, v=1.0471975511965976)
    $ 352 "C1mov_aprox" "breakAfter"
    movej(get_inverse_kin(pose_trans(C1mov_aprox_p, get_tcp_offset()), qnear=C1mov_aprox_q), a=1.3962634015954636, v=1.0471975511965976)
    $ 353 "MoveL"
    $ 354 "C1premove_3" "breakAfter"
    movel(pose_trans(pose_trans(Plane_3_C1move, pose_trans(p[-.180543022068, -.262061738902, .078420930934, 1.745866063160, .733967594413, 1.757652050583], C1premove_3_p)), get_tcp_offset()), a=0.6, v=0.08)
    $ 355 "MoveL"
    $ 356 "pl3C1mov_ini_1" "breakAfter"
    movel(pose_trans(Plane_3_C1move, pose_trans(p[-.180543022068, -.262061738902, .078420930934, 1.745866063160, .733967594413, 1.757652050583], pl3C1mov_ini_1_p)), a=0.6, v=0.08)
    $ 357 "Wait: 1.0"
    sleep(1.0)
    $ 358 "pl3C1mback_1" "breakAfter"
    movel(pose_trans(Plane_3_C1move, pose_trans(p[-.180543022068, -.262061738902, .078420930934, 1.745866063160, .733967594413, 1.757652050583], pl3C1mback_1_p)), a=0.6, v=0.08)
    $ 359 "pl3C1mback_ap_1" "breakAfter"
    movel(pose_trans(Plane_3_C1move, pose_trans(p[-.180543022068, -.262061738902, .078420930934, 1.745866063160, .733967594413, 1.757652050583], pl3C1mback_ap_1_p)), a=0.6, v=0.08)
    $ 360 "MoveJ"
    $ 361 "UL_C1mov_aprox" "breakAfter"
    movej(get_inverse_kin(UL_C1mov_aprox_p, qnear=UL_C1mov_aprox_q), a=1.3962634015954636, v=1.0471975511965976)
    $ 362 "UL_HomePos" "breakAfter"
    movej(get_inverse_kin(UL_HomePos_p, qnear=UL_HomePos_q), a=1.3962634015954636, v=1.0471975511965976)
  end
  def C2pk3move():
    $ 363 "C2pk3move" "noBreak"
    $ 364 "MoveJ"
    $ 365 "HomePos" "breakAfter"
    movej(get_inverse_kin(pose_trans(HomePos_p, get_tcp_offset()), qnear=HomePos_q), a=1.3962634015954636, v=1.0471975511965976)
    $ 366 "C2mov_aprox" "breakAfter"
    movej(get_inverse_kin(pose_trans(C2mov_aprox_p, get_tcp_offset()), qnear=C2mov_aprox_q), a=1.3962634015954636, v=1.0471975511965976)
    $ 367 "MoveL"
    $ 368 "C2premove_2" "breakAfter"
    movel(pose_trans(Plane_3_C1move, pose_trans(p[-.180543022068, -.262061738902, .078420930934, 1.745866063160, .733967594413, 1.757652050583], C2premove_2_p)), a=0.6, v=0.08)
    $ 369 "MoveL"
    $ 370 "pl3C2mov_ini_1" "breakAfter"
    movel(pose_trans(Plane_3_C1move, pose_trans(p[-.180543022068, -.262061738902, .078420930934, 1.745866063160, .733967594413, 1.757652050583], pl3C2mov_ini_1_p)), a=0.6, v=0.08)
    $ 371 "Wait: 1.0"
    sleep(1.0)
    $ 372 "pl3C2mback_1" "breakAfter"
    movel(pose_trans(Plane_3_C1move, pose_trans(p[-.180543022068, -.262061738902, .078420930934, 1.745866063160, .733967594413, 1.757652050583], pl3C2mback_1_p)), a=0.6, v=0.08)
    $ 373 "pl3C2mback_ap_1" "breakAfter"
    movel(pose_trans(Plane_3_C1move, pose_trans(p[-.180543022068, -.262061738902, .078420930934, 1.745866063160, .733967594413, 1.757652050583], pl3C2mback_ap_1_p)), a=0.6, v=0.08)
    $ 374 "MoveJ"
    $ 375 "C2mov_aprox" "breakAfter"
    movej(get_inverse_kin(pose_trans(C2mov_aprox_p, get_tcp_offset()), qnear=C2mov_aprox_q), a=1.3962634015954636, v=1.0471975511965976)
    $ 376 "HomePos" "breakAfter"
    movej(get_inverse_kin(pose_trans(HomePos_p, get_tcp_offset()), qnear=HomePos_q), a=1.3962634015954636, v=1.0471975511965976)
  end
  def C1pk4move():
    $ 377 "C1pk4move" "noBreak"
    $ 378 "MoveJ"
    $ 379 "HomePos" "breakAfter"
    movej(get_inverse_kin(pose_trans(HomePos_p, get_tcp_offset()), qnear=HomePos_q), a=1.3962634015954636, v=1.0471975511965976)
    $ 380 "C1mov_aprox" "breakAfter"
    movej(get_inverse_kin(pose_trans(C1mov_aprox_p, get_tcp_offset()), qnear=C1mov_aprox_q), a=1.3962634015954636, v=1.0471975511965976)
    $ 381 "MoveL"
    $ 382 "C1premove_4" "breakAfter"
    movel(pose_trans(Plane_3_C1move, pose_trans(p[-.180543022068, -.262061738902, .078420930934, 1.745866063160, .733967594413, 1.757652050583], C1premove_4_p)), a=0.6, v=0.08)
    $ 383 "MoveL"
    $ 384 "pl3C1mov_ini_2" "breakAfter"
    movel(pose_trans(Plane_3_C1move, pose_trans(p[-.180543022068, -.262061738902, .078420930934, 1.745866063160, .733967594413, 1.757652050583], pl3C1mov_ini_2_p)), a=0.6, v=0.08)
    $ 385 "Wait: 1.0"
    sleep(1.0)
    $ 386 "pl3C1mback_2" "breakAfter"
    movel(pose_trans(Plane_3_C1move, pose_trans(p[-.180543022068, -.262061738902, .078420930934, 1.745866063160, .733967594413, 1.757652050583], pl3C1mback_2_p)), a=0.6, v=0.08)
    $ 387 "pl3C1mback_ap_2" "breakAfter"
    movel(pose_trans(Plane_3_C1move, pose_trans(p[-.180543022068, -.262061738902, .078420930934, 1.745866063160, .733967594413, 1.757652050583], pl3C1mback_ap_2_p)), a=0.6, v=0.08)
    $ 388 "MoveJ"
    $ 389 "UL_C1mov_aprox" "breakAfter"
    movej(get_inverse_kin(UL_C1mov_aprox_p, qnear=UL_C1mov_aprox_q), a=1.3962634015954636, v=1.0471975511965976)
    $ 390 "UL_HomePos" "breakAfter"
    movej(get_inverse_kin(UL_HomePos_p, qnear=UL_HomePos_q), a=1.3962634015954636, v=1.0471975511965976)
  end
  def C2pk4move():
    $ 391 "C2pk4move" "noBreak"
    $ 392 "MoveJ"
    $ 393 "HomePos" "breakAfter"
    movej(get_inverse_kin(pose_trans(HomePos_p, get_tcp_offset()), qnear=HomePos_q), a=1.3962634015954636, v=1.0471975511965976)
    $ 394 "C2mov_aprox" "breakAfter"
    movej(get_inverse_kin(pose_trans(C2mov_aprox_p, get_tcp_offset()), qnear=C2mov_aprox_q), a=1.3962634015954636, v=1.0471975511965976)
    $ 395 "MoveL"
    $ 396 "C2premove_2" "breakAfter"
    movel(pose_trans(Plane_3_C1move, pose_trans(p[-.180543022068, -.262061738902, .078420930934, 1.745866063160, .733967594413, 1.757652050583], C2premove_2_p)), a=0.6, v=0.08)
    $ 397 "MoveL"
    $ 398 "pl3C2mov_ini_2" "breakAfter"
    movel(pose_trans(Plane_3_C1move, pose_trans(p[-.180543022068, -.262061738902, .078420930934, 1.745866063160, .733967594413, 1.757652050583], pl3C2mov_ini_2_p)), a=0.6, v=0.08)
    $ 399 "Wait: 1.0"
    sleep(1.0)
    $ 400 "pl3C2mback_2" "breakAfter"
    movel(pose_trans(Plane_3_C1move, pose_trans(p[-.180543022068, -.262061738902, .078420930934, 1.745866063160, .733967594413, 1.757652050583], pl3C2mback_2_p)), a=0.6, v=0.08)
    $ 401 "pl3C2mback_ap_2" "breakAfter"
    movel(pose_trans(Plane_3_C1move, pose_trans(p[-.180543022068, -.262061738902, .078420930934, 1.745866063160, .733967594413, 1.757652050583], pl3C2mback_ap_2_p)), a=0.6, v=0.08)
    $ 402 "MoveJ"
    $ 403 "C2mov_aprox" "breakAfter"
    movej(get_inverse_kin(pose_trans(C2mov_aprox_p, get_tcp_offset()), qnear=C2mov_aprox_q), a=1.3962634015954636, v=1.0471975511965976)
    $ 404 "HomePos" "breakAfter"
    movej(get_inverse_kin(pose_trans(HomePos_p, get_tcp_offset()), qnear=HomePos_q), a=1.3962634015954636, v=1.0471975511965976)
  end
  def C1pk5move():
    $ 405 "C1pk5move" "noBreak"
    $ 406 "MoveJ"
    $ 407 "UL_HomePos" "breakAfter"
    movej(get_inverse_kin(UL_HomePos_p, qnear=UL_HomePos_q), a=1.3962634015954636, v=1.0471975511965976)
    $ 408 "UL_C1mov_aprox" "breakAfter"
    movej(get_inverse_kin(UL_C1mov_aprox_p, qnear=UL_C1mov_aprox_q), a=1.3962634015954636, v=1.0471975511965976)
    $ 409 "MoveL"
    $ 410 "C1premove_5" "breakAfter"
    movel(pose_trans(Plane_3_C1move, pose_trans(p[-.180543022068, -.262061738902, .078420930934, 1.745866063160, .733967594413, 1.757652050583], C1premove_5_p)), a=0.6, v=0.08)
    $ 411 "MoveL"
    $ 412 "pl3C1mov_ini_3" "breakAfter"
    movel(pose_trans(Plane_3_C1move, pose_trans(p[-.180543022068, -.262061738902, .078420930934, 1.745866063160, .733967594413, 1.757652050583], pl3C1mov_ini_3_p)), a=0.6, v=0.08)
    $ 413 "Wait: 1.0"
    sleep(1.0)
    $ 414 "pl3C1mback_3" "breakAfter"
    movel(pose_trans(Plane_3_C1move, pose_trans(p[-.180543022068, -.262061738902, .078420930934, 1.745866063160, .733967594413, 1.757652050583], pl3C1mback_3_p)), a=0.6, v=0.08)
    $ 415 "pl3C1mback_ap_3" "breakAfter"
    movel(pose_trans(Plane_3_C1move, pose_trans(p[-.180543022068, -.262061738902, .078420930934, 1.745866063160, .733967594413, 1.757652050583], pl3C1mback_ap_3_p)), a=0.6, v=0.08)
    $ 416 "MoveJ"
    $ 417 "UL_C1mov_aprox" "breakAfter"
    movej(get_inverse_kin(UL_C1mov_aprox_p, qnear=UL_C1mov_aprox_q), a=1.3962634015954636, v=1.0471975511965976)
    $ 418 "UL_HomePos" "breakAfter"
    movej(get_inverse_kin(UL_HomePos_p, qnear=UL_HomePos_q), a=1.3962634015954636, v=1.0471975511965976)
  end
  def C2pk5move():
    $ 419 "C2pk5move" "noBreak"
    $ 420 "MoveJ"
    $ 421 "HomePos" "breakAfter"
    movej(get_inverse_kin(pose_trans(HomePos_p, get_tcp_offset()), qnear=HomePos_q), a=1.3962634015954636, v=1.0471975511965976)
    $ 422 "C2mov_aprox" "breakAfter"
    movej(get_inverse_kin(pose_trans(C2mov_aprox_p, get_tcp_offset()), qnear=C2mov_aprox_q), a=1.3962634015954636, v=1.0471975511965976)
    $ 423 "MoveL"
    $ 424 "C2premove_2" "breakAfter"
    movel(pose_trans(Plane_3_C1move, pose_trans(p[-.180543022068, -.262061738902, .078420930934, 1.745866063160, .733967594413, 1.757652050583], C2premove_2_p)), a=0.6, v=0.08)
    $ 425 "MoveL"
    $ 426 "pl3C2mov_ini_3" "breakAfter"
    movel(pose_trans(Plane_3_C1move, pose_trans(p[-.180543022068, -.262061738902, .078420930934, 1.745866063160, .733967594413, 1.757652050583], pl3C2mov_ini_3_p)), a=0.6, v=0.08)
    $ 427 "Wait: 1.0"
    sleep(1.0)
    $ 428 "pl3C2mback_3" "breakAfter"
    movel(pose_trans(Plane_3_C1move, pose_trans(p[-.180543022068, -.262061738902, .078420930934, 1.745866063160, .733967594413, 1.757652050583], pl3C2mback_3_p)), a=0.6, v=0.08)
    $ 429 "pl3C2mback_ap_3" "breakAfter"
    movel(pose_trans(Plane_3_C1move, pose_trans(p[-.180543022068, -.262061738902, .078420930934, 1.745866063160, .733967594413, 1.757652050583], pl3C2mback_ap_3_p)), a=0.6, v=0.08)
    $ 430 "MoveJ"
    $ 431 "C2mov_aprox" "breakAfter"
    movej(get_inverse_kin(pose_trans(C2mov_aprox_p, get_tcp_offset()), qnear=C2mov_aprox_q), a=1.3962634015954636, v=1.0471975511965976)
    $ 432 "HomePos" "breakAfter"
    movej(get_inverse_kin(pose_trans(HomePos_p, get_tcp_offset()), qnear=HomePos_q), a=1.3962634015954636, v=1.0471975511965976)
  end
  def PACK1_pick():
    $ 433 "PACK1_pick" "noBreak"
    $ 434 "Set OutNet_Tool=Off"
    write_output_boolean_register(2, False)
    $ 435 "Set OuTNET_Gripper=0"
    write_output_integer_register(0, 0)
    $ 436 "Wait: 1.0"
    sleep(1.0)
    $ 437 "Set OutNet_Tool=On"
    write_output_boolean_register(2, True)
    $ 438 "Wait: 2.0"
    sleep(2.0)
    $ 439 "MoveJ"
    $ 440 "UL_HomePos" "breakAfter"
    movej(get_inverse_kin(UL_HomePos_p, qnear=UL_HomePos_q), a=1.3962634015954636, v=1.0471975511965976)
    $ 441 "Set OutNet_Tool=Off"
    write_output_boolean_register(2, False)
    $ 442 "UL_Pack_aprox_1" "breakAfter"
    movej(get_inverse_kin(UL_Pack_aprox_1_p, qnear=UL_Pack_aprox_1_q), a=1.3962634015954636, v=1.0471975511965976)
    $ 443 "MoveL"
    $ 444 "pl1_PK1up_2" "breakAfter"
    movel(pose_trans(Plane_1_Pack, pose_trans(p[.061451264231, -.289311417922, -.073379282729, -.000157706105, .000169116670, 2.356123162082], pl1_PK1up_2_p)), a=1.2, v=0.25)
    $ 445 "MoveL"
    $ 446 "pl1_PK1_1" "breakAfter"
    movel(pose_trans(Plane_1_Pack, pose_trans(p[.061451264231, -.289311417922, -.073379282729, -.000157706105, .000169116670, 2.356123162082], pl1_PK1_1_p)), a=1.2, v=0.25)
    $ 447 "Set OuTNET_Gripper=5"
    write_output_integer_register(0, 5)
    $ 448 "Set OutNet_Tool=On"
    write_output_boolean_register(2, True)
    $ 449 "Wait: 5.0"
    sleep(5.0)
    $ 450 "Wait InNET_InPos=HI"
    while (read_input_boolean_register(1) == False):
      sync()
    end
    $ 451 "Set OutNet_Tool=Off"
    write_output_boolean_register(2, False)
    $ 452 "pl1_PK1up_3" "breakAfter"
    movel(pose_trans(Plane_1_Pack, pose_trans(p[.061451264231, -.289311417922, -.073379282729, -.000157706105, .000169116670, 2.356123162082], pl1_PK1up_3_p)), a=1.2, v=0.25)
    $ 453 "MoveJ"
    $ 454 "UL_Pack_aprox_1" "breakAfter"
    movej(get_inverse_kin(UL_Pack_aprox_1_p, qnear=UL_Pack_aprox_1_q), a=1.3962634015954636, v=1.0471975511965976)
  end
  def PACK2_pick():
    $ 455 "PACK2_pick" "noBreak"
    $ 456 "MoveJ"
    $ 457 "UL_HomePos" "breakAfter"
    movej(get_inverse_kin(UL_HomePos_p, qnear=UL_HomePos_q), a=1.3962634015954636, v=1.0471975511965976)
    $ 458 "Set OutNet_Tool=Off"
    write_output_boolean_register(2, False)
    $ 459 "Set OutNET_Done=Off"
    write_output_boolean_register(1, False)
    $ 460 "UL_Pack_aprox_1" "breakAfter"
    movej(get_inverse_kin(UL_Pack_aprox_1_p, qnear=UL_Pack_aprox_1_q), a=1.3962634015954636, v=1.0471975511965976)
    $ 461 "MoveL"
    $ 462 "pl1_PK2up_2" "breakAfter"
    movel(pose_trans(Plane_1_Pack, pose_trans(p[.061451264231, -.289311417922, -.073379282729, -.000157706105, .000169116670, 2.356123162082], pl1_PK2up_2_p)), a=1.2, v=0.25)
    $ 463 "MoveL"
    $ 464 "p1_PK2_1" "breakAfter"
    movel(pose_trans(Plane_1_Pack, pose_trans(p[.061451264231, -.289311417922, -.073379282729, -.000157706105, .000169116670, 2.356123162082], p1_PK2_1_p)), a=1.2, v=0.25)
    $ 465 "Set OuTNET_Gripper=5"
    write_output_integer_register(0, 5)
    $ 466 "Set OutNet_Tool=On"
    write_output_boolean_register(2, True)
    $ 467 "Wait: 2.0"
    sleep(2.0)
    $ 468 "Wait: 5.0"
    sleep(5.0)
    $ 469 "Set OutNet_Tool=Off"
    write_output_boolean_register(2, False)
    $ 470 "pl1_PK2up_3" "breakAfter"
    movel(pose_trans(Plane_1_Pack, pose_trans(p[.061451264231, -.289311417922, -.073379282729, -.000157706105, .000169116670, 2.356123162082], pl1_PK2up_3_p)), a=1.2, v=0.25)
    $ 471 "MoveJ"
    $ 472 "UL_Pack_aprox_1" "breakAfter"
    movej(get_inverse_kin(UL_Pack_aprox_1_p, qnear=UL_Pack_aprox_1_q), a=1.3962634015954636, v=1.0471975511965976)
  end
  def PACK3_pick():
    $ 473 "PACK3_pick" "noBreak"
    $ 474 "Set OutNet_Tool=Off"
    write_output_boolean_register(2, False)
    $ 475 "MoveJ"
    $ 476 "UL_HomePos" "breakAfter"
    movej(get_inverse_kin(UL_HomePos_p, qnear=UL_HomePos_q), a=1.3962634015954636, v=1.0471975511965976)
    $ 477 "UL_Pack_aprox_1" "breakAfter"
    movej(get_inverse_kin(UL_Pack_aprox_1_p, qnear=UL_Pack_aprox_1_q), a=1.3962634015954636, v=1.0471975511965976)
    $ 478 "Set OuTNET_Gripper=0"
    write_output_integer_register(0, 0)
    $ 479 "Set OutNet_Tool=On"
    write_output_boolean_register(2, True)
    $ 480 "MoveL"
    $ 481 "pl1_PK3up_2" "breakAfter"
    movel(pose_trans(Plane_1_Pack, pose_trans(p[.061451264231, -.289311417922, -.073379282729, -.000157706105, .000169116670, 2.356123162082], pl1_PK3up_2_p)), a=1.2, v=0.25)
    $ 482 "Wait: 1.0"
    sleep(1.0)
    $ 483 "Set OutNet_Tool=Off"
    write_output_boolean_register(2, False)
    $ 484 "MoveL"
    $ 485 "pl1_PK3_1" "breakAfter"
    movel(pose_trans(Plane_1_Pack, pose_trans(p[.061451264231, -.289311417922, -.073379282729, -.000157706105, .000169116670, 2.356123162082], pl1_PK3_1_p)), a=1.2, v=0.25)
    $ 486 "Wait: 1.0"
    sleep(1.0)
    $ 487 "Set OuTNET_Gripper=5"
    write_output_integer_register(0, 5)
    $ 488 "Set OutNet_Tool=On"
    write_output_boolean_register(2, True)
    $ 489 "Wait: 5.0"
    sleep(5.0)
    $ 490 "pl1_PK3up_3" "breakAfter"
    movel(pose_trans(Plane_1_Pack, pose_trans(p[.061451264231, -.289311417922, -.073379282729, -.000157706105, .000169116670, 2.356123162082], pl1_PK3up_3_p)), a=1.2, v=0.25)
    $ 491 "MoveJ"
    $ 492 "UL_Pack_aprox_1" "breakAfter"
    movej(get_inverse_kin(UL_Pack_aprox_1_p, qnear=UL_Pack_aprox_1_q), a=1.3962634015954636, v=1.0471975511965976)
  end
  def PACK_Unload():
    $ 493 "PACK_Unload" "noBreak"
    $ 494 "MoveJ"
    $ 495 "Belt_up" "breakAfter"
    movej(get_inverse_kin(Belt_up_p, qnear=Belt_up_q), a=1.3962634015954636, v=1.0471975511965976)
    $ 496 "MoveL"
    $ 497 "Belt_end" "breakAfter"
    movel(pose_trans(Belt_end_p, get_tcp_offset()), a=1.2, v=0.25, r=0.01)
    $ 498 "Belt_down" "breakAfter"
    movel(pose_trans(Belt_down_p, get_tcp_offset()), a=1.2, v=0.25)
    $ 499 "Set OutNet_Tool=Off"
    write_output_boolean_register(2, False)
    $ 500 "Wait: 1.0"
    sleep(1.0)
    $ 501 "Set OuTNET_Gripper=0"
    write_output_integer_register(0, 0)
    $ 502 "Set OutNet_Tool=On"
    write_output_boolean_register(2, True)
    $ 503 "Wait: 2.0"
    sleep(2.0)
    $ 504 "Wait InNET_InPos=HI"
    while (read_input_boolean_register(1) == False):
      sync()
    end
    $ 505 "Set OutNet_Tool=Off"
    write_output_boolean_register(2, False)
    $ 506 "Belt_end" "breakAfter"
    movel(pose_trans(Belt_end_p, get_tcp_offset()), a=1.2, v=0.25)
    $ 507 "Wait: 1.0"
    sleep(1.0)
    $ 508 "Set OuTNET_Gripper=8"
    write_output_integer_register(0, 8)
    $ 509 "Set OutNet_Tool=On"
    write_output_boolean_register(2, True)
    $ 510 "Wait: 5.0"
    sleep(5.0)
    $ 511 "MoveJ"
    $ 512 "HomePos" "breakAfter"
    movej(get_inverse_kin(pose_trans(HomePos_p, get_tcp_offset()), qnear=HomePos_q), a=1.3962634015954636, v=1.0471975511965976)
  end
  def PALLET__remove():
    $ 513 "PALLET__remove" "noBreak"
    $ 514 "MoveJ"
    $ 515 "Pallet_prepick" "breakAfter"
    movej(get_inverse_kin(pose_trans(Pallet_prepick_p, get_tcp_offset()), qnear=Pallet_prepick_q), a=1.3962634015954636, v=1.0471975511965976)
    $ 516 "MoveL"
    $ 517 "Pallet_pick" "breakAfter"
    movel(pose_trans(Pallet_pick_p, get_tcp_offset()), a=1.2, v=0.25)
    $ 518 "Set OuTNET_Gripper=5"
    write_output_integer_register(0, 5)
    $ 519 "Set OutNet_Tool=On"
    write_output_boolean_register(2, True)
    $ 520 "Wait: 3.0"
    sleep(3.0)
    $ 521 "Wait InNET_InPos=HI"
    while (read_input_boolean_register(1) == False):
      sync()
    end
    $ 522 "Set OutNet_Tool=Off"
    write_output_boolean_register(2, False)
    $ 523 "Pallet_prepick" "breakAfter"
    movel(pose_trans(Pallet_prepick_p, get_tcp_offset()), a=1.2, v=0.25)
    $ 524 "Pallet_release" "breakAfter"
    movel(pose_trans(Pallet_release_p, get_tcp_offset()), a=1.2, v=0.25)
    $ 525 "If InNET_PalletNum≠1 and InNET_PalletNum≠3 and InNET_PalletNum≠5 and InNET_PalletNum≠7"
    if (read_input_integer_register(1) != 1  and  read_input_integer_register(1) != 3  and  read_input_integer_register(1) != 5  and  read_input_integer_register(1) != 7):
      $ 526 "If InNET_PalletNum≤5"
      if (read_input_integer_register(1) <= 5):
        $ 527 "D1_pallet_down" "breakAfter"
        movel(pose_trans(D1_pallet_down_p, get_tcp_offset()), a=1.2, v=0.25)
      else:
        $ 528 "Else" "noBreak"
        $ 529 "D1_pallet_up" "breakAfter"
        movel(pose_trans(D1_pallet_up_p, get_tcp_offset()), a=1.2, v=0.25)
      end
    else:
      $ 530 "ElseIf InNET_PalletNum≤5"
      if (read_input_integer_register(1) <= 5):
        $ 531 "D2_pallet_down" "breakAfter"
        movel(pose_trans(D2_pallet_down_p, get_tcp_offset()), a=1.2, v=0.25)
      else:
        $ 532 "Else" "noBreak"
        $ 533 "D2_pallet_up" "breakAfter"
        movel(pose_trans(D2_pallet_up_p, get_tcp_offset()), a=1.2, v=0.25)
      end
    end
    $ 534 "Set OuTNET_Gripper=0"
    write_output_integer_register(0, 0)
    $ 535 "Set OutNet_Tool=On"
    write_output_boolean_register(2, True)
    $ 536 "Wait: 3.0"
    sleep(3.0)
    $ 537 "Wait InNET_InPos=HI"
    while (read_input_boolean_register(1) == False):
      sync()
    end
    $ 538 "Set OutNet_Tool=Off"
    write_output_boolean_register(2, False)
    $ 539 "D_UP" "breakAfter"
    movel(pose_trans(D_UP_p, get_tcp_offset()), a=1.2, v=0.25)
    $ 540 "If InNET_PalletNum≥8"
    if (read_input_integer_register(1) >= 8):
      $ 541 "MoveJ"
      $ 542 "HomePos" "breakAfter"
      movej(get_inverse_kin(pose_trans(HomePos_p, get_tcp_offset()), qnear=HomePos_q), a=1.3962634015954636, v=1.0471975511965976)
      $ 543 "Set OutNet_FullBin=On"
      write_output_boolean_register(3, True)
      $ 544 "Wait: 2.0"
      sleep(2.0)
      $ 545 "Set OutNet_FullBin=Off"
      write_output_boolean_register(3, False)
      $ 546 "Wait: 2.0"
      sleep(2.0)
      $ 547 "Wait InNET_Enable"
      while (not(read_input_boolean_register(2))):
        sync()
      end
    else:
      $ 548 "Else" "noBreak"
      $ 549 "MoveJ"
      $ 550 "HomePos" "breakAfter"
      movej(get_inverse_kin(pose_trans(HomePos_p, get_tcp_offset()), qnear=HomePos_q), a=1.3962634015954636, v=1.0471975511965976)
    end
  end
  def PK1CAN1_release():
    $ 551 "PK1CAN1_release" "noBreak"
    $ 552 "MoveJ"
    $ 553 "Pallet_prepick" "breakAfter"
    movej(get_inverse_kin(pose_trans(Pallet_prepick_p, get_tcp_offset()), qnear=Pallet_prepick_q), a=1.3962634015954636, v=1.0471975511965976)
    $ 554 "MoveL"
    $ 555 "Pick_canister" "breakAfter"
    movel(pose_trans(Pick_canister_p, get_tcp_offset()), a=1.2, v=0.25)
    $ 556 "Set OuTNET_Gripper=6"
    write_output_integer_register(0, 6)
    $ 557 "Set OutNet_Tool=On"
    write_output_boolean_register(2, True)
    $ 558 "Wait: 3.0"
    sleep(3.0)
    $ 559 "Wait InNET_InPos=HI"
    while (read_input_boolean_register(1) == False):
      sync()
    end
    $ 560 "Set OutNet_Tool=Off"
    write_output_boolean_register(2, False)
    $ 561 "MoveL"
    $ 562 "Pallet_prepick" "breakAfter"
    movel(pose_trans(Pallet_prepick_p, get_tcp_offset()), a=1.2, v=0.25)
    $ 563 "MoveJ"
    $ 564 "Canister_aprox" "breakAfter"
    movej(get_inverse_kin(Canister_aprox_p, qnear=Canister_aprox_q), a=1.3962634015954636, v=1.0471975511965976)
    $ 565 "MoveL"
    $ 566 "pl1Canister11up" "breakAfter"
    movel(pose_trans(Plane_1_Pack, pose_trans(p[.061451264231, -.289311417922, -.073379282729, -.000157706105, .000169116670, 2.356123162082], pl1Canister11up_p)), a=1.2, v=0.25)
    $ 567 "MoveL"
    $ 568 "pl1Canister11" "breakAfter"
    movel(pose_trans(Plane_1_Pack, pose_trans(p[.061451264231, -.289311417922, -.073379282729, -.000157706105, .000169116670, 2.356123162082], pl1Canister11_p)), a=1.2, v=0.25)
    $ 569 "Set OuTNET_Gripper=2"
    write_output_integer_register(0, 2)
    $ 570 "Set OutNet_Tool=On"
    write_output_boolean_register(2, True)
    $ 571 "Wait: 3.0"
    sleep(3.0)
    $ 572 "Wait InNET_InPos=HI"
    while (read_input_boolean_register(1) == False):
      sync()
    end
    $ 573 "Set OutNet_Tool=Off"
    write_output_boolean_register(2, False)
    $ 574 "MoveL"
    $ 575 "pl1Canist11up_1" "breakAfter"
    movel(pose_trans(Plane_1_Pack, pose_trans(p[.061451264231, -.289311417922, -.073379282729, -.000157706105, .000169116670, 2.356123162082], pl1Canist11up_1_p)), a=1.2, v=0.25)
    $ 576 "MoveJ"
    $ 577 "Canister_aprox" "breakAfter"
    movej(get_inverse_kin(Canister_aprox_p, qnear=Canister_aprox_q), a=1.3962634015954636, v=1.0471975511965976)
  end
  def PK1CAN2_release():
    $ 578 "PK1CAN2_release" "noBreak"
    $ 579 "MoveJ"
    $ 580 "Pallet_prepick" "breakAfter"
    movej(get_inverse_kin(pose_trans(Pallet_prepick_p, get_tcp_offset()), qnear=Pallet_prepick_q), a=1.3962634015954636, v=1.0471975511965976)
    $ 581 "MoveL"
    $ 582 "Pick_canister" "breakAfter"
    movel(pose_trans(Pick_canister_p, get_tcp_offset()), a=1.2, v=0.25)
    $ 583 "Set OuTNET_Gripper=6"
    write_output_integer_register(0, 6)
    $ 584 "Set OutNet_Tool=On"
    write_output_boolean_register(2, True)
    $ 585 "Wait: 3.0"
    sleep(3.0)
    $ 586 "Wait InNET_InPos=HI"
    while (read_input_boolean_register(1) == False):
      sync()
    end
    $ 587 "Set OutNet_Tool=Off"
    write_output_boolean_register(2, False)
    $ 588 "MoveL"
    $ 589 "Pallet_prepick" "breakAfter"
    movel(pose_trans(Pallet_prepick_p, get_tcp_offset()), a=1.2, v=0.25)
    $ 590 "MoveJ"
    $ 591 "Canister_aprox" "breakAfter"
    movej(get_inverse_kin(Canister_aprox_p, qnear=Canister_aprox_q), a=1.3962634015954636, v=1.0471975511965976)
    $ 592 "MoveL"
    $ 593 "pl1Canister12up" "breakAfter"
    movel(pose_trans(Plane_1_Pack, pose_trans(p[.061451264231, -.289311417922, -.073379282729, -.000157706105, .000169116670, 2.356123162082], pl1Canister12up_p)), a=1.2, v=0.25)
    $ 594 "MoveL"
    $ 595 "pl1Canister12" "breakAfter"
    movel(pose_trans(Plane_1_Pack, pose_trans(p[.061451264231, -.289311417922, -.073379282729, -.000157706105, .000169116670, 2.356123162082], pl1Canister12_p)), a=1.2, v=0.25)
    $ 596 "Set OuTNET_Gripper=2"
    write_output_integer_register(0, 2)
    $ 597 "Set OutNet_Tool=On"
    write_output_boolean_register(2, True)
    $ 598 "Wait: 3.0"
    sleep(3.0)
    $ 599 "Wait InNET_InPos=HI"
    while (read_input_boolean_register(1) == False):
      sync()
    end
    $ 600 "Set OutNet_Tool=Off"
    write_output_boolean_register(2, False)
    $ 601 "MoveL"
    $ 602 "pl1Canist12up" "breakAfter"
    movel(pose_trans(Plane_1_Pack, pose_trans(p[.061451264231, -.289311417922, -.073379282729, -.000157706105, .000169116670, 2.356123162082], pl1Canist12up_p)), a=1.2, v=0.25)
    $ 603 "MoveJ"
    $ 604 "Canister_aprox" "breakAfter"
    movej(get_inverse_kin(Canister_aprox_p, qnear=Canister_aprox_q), a=1.3962634015954636, v=1.0471975511965976)
  end
  def PK1CAN3_release():
    $ 605 "PK1CAN3_release" "noBreak"
    $ 606 "MoveJ"
    $ 607 "Pallet_prepick" "breakAfter"
    movej(get_inverse_kin(pose_trans(Pallet_prepick_p, get_tcp_offset()), qnear=Pallet_prepick_q), a=1.3962634015954636, v=1.0471975511965976)
    $ 608 "MoveL"
    $ 609 "Pick_canister" "breakAfter"
    movel(pose_trans(Pick_canister_p, get_tcp_offset()), a=1.2, v=0.25)
    $ 610 "Set OuTNET_Gripper=6"
    write_output_integer_register(0, 6)
    $ 611 "Set OutNet_Tool=On"
    write_output_boolean_register(2, True)
    $ 612 "Wait: 3.0"
    sleep(3.0)
    $ 613 "Wait InNET_InPos=HI"
    while (read_input_boolean_register(1) == False):
      sync()
    end
    $ 614 "Set OutNet_Tool=Off"
    write_output_boolean_register(2, False)
    $ 615 "MoveL"
    $ 616 "Pallet_prepick" "breakAfter"
    movel(pose_trans(Pallet_prepick_p, get_tcp_offset()), a=1.2, v=0.25)
    $ 617 "MoveJ"
    $ 618 "Canister_aprox" "breakAfter"
    movej(get_inverse_kin(Canister_aprox_p, qnear=Canister_aprox_q), a=1.3962634015954636, v=1.0471975511965976)
    $ 619 "MoveL"
    $ 620 "pl1Canister13up" "breakAfter"
    movel(pose_trans(Plane_1_Pack, pose_trans(p[.061451264231, -.289311417922, -.073379282729, -.000157706105, .000169116670, 2.356123162082], pl1Canister13up_p)), a=1.2, v=0.25)
    $ 621 "MoveL"
    $ 622 "pl1Canister13" "breakAfter"
    movel(pose_trans(Plane_1_Pack, pose_trans(p[.061451264231, -.289311417922, -.073379282729, -.000157706105, .000169116670, 2.356123162082], pl1Canister13_p)), a=1.2, v=0.25)
    $ 623 "Set OuTNET_Gripper=2"
    write_output_integer_register(0, 2)
    $ 624 "Set OutNet_Tool=On"
    write_output_boolean_register(2, True)
    $ 625 "Wait: 3.0"
    sleep(3.0)
    $ 626 "Wait InNET_InPos=HI"
    while (read_input_boolean_register(1) == False):
      sync()
    end
    $ 627 "Set OutNet_Tool=Off"
    write_output_boolean_register(2, False)
    $ 628 "MoveL"
    $ 629 "pl1Canist13up" "breakAfter"
    movel(pose_trans(Plane_1_Pack, pose_trans(p[.061451264231, -.289311417922, -.073379282729, -.000157706105, .000169116670, 2.356123162082], pl1Canist13up_p)), a=1.2, v=0.25)
    $ 630 "MoveJ"
    $ 631 "Canister_aprox" "breakAfter"
    movej(get_inverse_kin(Canister_aprox_p, qnear=Canister_aprox_q), a=1.3962634015954636, v=1.0471975511965976)
  end
  def PK1CAN4_release():
    $ 632 "PK1CAN4_release" "noBreak"
    $ 633 "MoveJ"
    $ 634 "Pallet_prepick" "breakAfter"
    movej(get_inverse_kin(pose_trans(Pallet_prepick_p, get_tcp_offset()), qnear=Pallet_prepick_q), a=1.3962634015954636, v=1.0471975511965976)
    $ 635 "MoveL"
    $ 636 "Pick_canister" "breakAfter"
    movel(pose_trans(Pick_canister_p, get_tcp_offset()), a=1.2, v=0.25)
    $ 637 "Set OuTNET_Gripper=6"
    write_output_integer_register(0, 6)
    $ 638 "Set OutNet_Tool=On"
    write_output_boolean_register(2, True)
    $ 639 "Wait: 3.0"
    sleep(3.0)
    $ 640 "Wait InNET_InPos=HI"
    while (read_input_boolean_register(1) == False):
      sync()
    end
    $ 641 "Set OutNet_Tool=Off"
    write_output_boolean_register(2, False)
    $ 642 "MoveL"
    $ 643 "Pallet_prepick" "breakAfter"
    movel(pose_trans(Pallet_prepick_p, get_tcp_offset()), a=1.2, v=0.25)
    $ 644 "MoveJ"
    $ 645 "Canister_aprox" "breakAfter"
    movej(get_inverse_kin(Canister_aprox_p, qnear=Canister_aprox_q), a=1.3962634015954636, v=1.0471975511965976)
    $ 646 "MoveL"
    $ 647 "pl1Canister14up" "breakAfter"
    movel(pose_trans(Plane_1_Pack, pose_trans(p[.061451264231, -.289311417922, -.073379282729, -.000157706105, .000169116670, 2.356123162082], pl1Canister14up_p)), a=1.2, v=0.25)
    $ 648 "MoveL"
    $ 649 "pl1Canister14" "breakAfter"
    movel(pose_trans(Plane_1_Pack, pose_trans(p[.061451264231, -.289311417922, -.073379282729, -.000157706105, .000169116670, 2.356123162082], pl1Canister14_p)), a=1.2, v=0.25)
    $ 650 "Set OuTNET_Gripper=2"
    write_output_integer_register(0, 2)
    $ 651 "Set OutNet_Tool=On"
    write_output_boolean_register(2, True)
    $ 652 "Wait: 3.0"
    sleep(3.0)
    $ 653 "Wait InNET_InPos=HI"
    while (read_input_boolean_register(1) == False):
      sync()
    end
    $ 654 "Set OutNet_Tool=Off"
    write_output_boolean_register(2, False)
    $ 655 "MoveL"
    $ 656 "pl1Canist14up" "breakAfter"
    movel(pose_trans(Plane_1_Pack, pose_trans(p[.061451264231, -.289311417922, -.073379282729, -.000157706105, .000169116670, 2.356123162082], pl1Canist14up_p)), a=1.2, v=0.25)
    $ 657 "MoveJ"
    $ 658 "Canister_aprox" "breakAfter"
    movej(get_inverse_kin(Canister_aprox_p, qnear=Canister_aprox_q), a=1.3962634015954636, v=1.0471975511965976)
  end
  def PK2CAN1_release():
    $ 659 "PK2CAN1_release" "noBreak"
    $ 660 "MoveJ"
    $ 661 "Pallet_prepick" "breakAfter"
    movej(get_inverse_kin(pose_trans(Pallet_prepick_p, get_tcp_offset()), qnear=Pallet_prepick_q), a=1.3962634015954636, v=1.0471975511965976)
    $ 662 "MoveL"
    $ 663 "Pick_canister" "breakAfter"
    movel(pose_trans(Pick_canister_p, get_tcp_offset()), a=1.2, v=0.25)
    $ 664 "Set OuTNET_Gripper=6"
    write_output_integer_register(0, 6)
    $ 665 "Set OutNet_Tool=On"
    write_output_boolean_register(2, True)
    $ 666 "Wait: 3.0"
    sleep(3.0)
    $ 667 "Wait InNET_InPos=HI"
    while (read_input_boolean_register(1) == False):
      sync()
    end
    $ 668 "Set OutNet_Tool=Off"
    write_output_boolean_register(2, False)
    $ 669 "MoveL"
    $ 670 "Pallet_prepick" "breakAfter"
    movel(pose_trans(Pallet_prepick_p, get_tcp_offset()), a=1.2, v=0.25)
    $ 671 "MoveJ"
    $ 672 "Canister_aprox" "breakAfter"
    movej(get_inverse_kin(Canister_aprox_p, qnear=Canister_aprox_q), a=1.3962634015954636, v=1.0471975511965976)
    $ 673 "MoveL"
    $ 674 "pl1Canister21up" "breakAfter"
    movel(pose_trans(Plane_1_Pack, pose_trans(p[.061451264231, -.289311417922, -.073379282729, -.000157706105, .000169116670, 2.356123162082], pl1Canister21up_p)), a=1.2, v=0.25)
    $ 675 "MoveL"
    $ 676 "pl1Canister21" "breakAfter"
    movel(pose_trans(Plane_1_Pack, pose_trans(p[.061451264231, -.289311417922, -.073379282729, -.000157706105, .000169116670, 2.356123162082], pl1Canister21_p)), a=1.2, v=0.25)
    $ 677 "Set OuTNET_Gripper=2"
    write_output_integer_register(0, 2)
    $ 678 "Set OutNet_Tool=On"
    write_output_boolean_register(2, True)
    $ 679 "Wait: 3.0"
    sleep(3.0)
    $ 680 "Wait InNET_InPos=HI"
    while (read_input_boolean_register(1) == False):
      sync()
    end
    $ 681 "Set OutNet_Tool=Off"
    write_output_boolean_register(2, False)
    $ 682 "MoveL"
    $ 683 "pl1Canist21up" "breakAfter"
    movel(pose_trans(Plane_1_Pack, pose_trans(p[.061451264231, -.289311417922, -.073379282729, -.000157706105, .000169116670, 2.356123162082], pl1Canist21up_p)), a=1.2, v=0.25)
    $ 684 "MoveJ"
    $ 685 "Canister_aprox" "breakAfter"
    movej(get_inverse_kin(Canister_aprox_p, qnear=Canister_aprox_q), a=1.3962634015954636, v=1.0471975511965976)
  end
  def PK2CAN2_release():
    $ 686 "PK2CAN2_release" "noBreak"
    $ 687 "MoveJ"
    $ 688 "Pallet_prepick" "breakAfter"
    movej(get_inverse_kin(pose_trans(Pallet_prepick_p, get_tcp_offset()), qnear=Pallet_prepick_q), a=1.3962634015954636, v=1.0471975511965976)
    $ 689 "MoveL"
    $ 690 "Pick_canister" "breakAfter"
    movel(pose_trans(Pick_canister_p, get_tcp_offset()), a=1.2, v=0.25)
    $ 691 "Set OuTNET_Gripper=6"
    write_output_integer_register(0, 6)
    $ 692 "Set OutNet_Tool=On"
    write_output_boolean_register(2, True)
    $ 693 "Wait: 3.0"
    sleep(3.0)
    $ 694 "Wait InNET_InPos=HI"
    while (read_input_boolean_register(1) == False):
      sync()
    end
    $ 695 "Set OutNet_Tool=Off"
    write_output_boolean_register(2, False)
    $ 696 "MoveL"
    $ 697 "Pallet_prepick" "breakAfter"
    movel(pose_trans(Pallet_prepick_p, get_tcp_offset()), a=1.2, v=0.25)
    $ 698 "MoveJ"
    $ 699 "Canister_aprox" "breakAfter"
    movej(get_inverse_kin(Canister_aprox_p, qnear=Canister_aprox_q), a=1.3962634015954636, v=1.0471975511965976)
    $ 700 "MoveL"
    $ 701 "pl1Canister22up" "breakAfter"
    movel(pose_trans(Plane_1_Pack, pose_trans(p[.061451264231, -.289311417922, -.073379282729, -.000157706105, .000169116670, 2.356123162082], pl1Canister22up_p)), a=1.2, v=0.25)
    $ 702 "MoveL"
    $ 703 "pl1Canister22" "breakAfter"
    movel(pose_trans(Plane_1_Pack, pose_trans(p[.061451264231, -.289311417922, -.073379282729, -.000157706105, .000169116670, 2.356123162082], pl1Canister22_p)), a=1.2, v=0.25)
    $ 704 "Set OuTNET_Gripper=2"
    write_output_integer_register(0, 2)
    $ 705 "Set OutNet_Tool=On"
    write_output_boolean_register(2, True)
    $ 706 "Wait: 3.0"
    sleep(3.0)
    $ 707 "Wait InNET_InPos=HI"
    while (read_input_boolean_register(1) == False):
      sync()
    end
    $ 708 "Set OutNet_Tool=Off"
    write_output_boolean_register(2, False)
    $ 709 "MoveL"
    $ 710 "pl1Canist22up" "breakAfter"
    movel(pose_trans(Plane_1_Pack, pose_trans(p[.061451264231, -.289311417922, -.073379282729, -.000157706105, .000169116670, 2.356123162082], pl1Canist22up_p)), a=1.2, v=0.25)
    $ 711 "MoveJ"
    $ 712 "Canister_aprox" "breakAfter"
    movej(get_inverse_kin(Canister_aprox_p, qnear=Canister_aprox_q), a=1.3962634015954636, v=1.0471975511965976)
  end
  def PK2CAN3_release():
    $ 713 "PK2CAN3_release" "noBreak"
    $ 714 "MoveJ"
    $ 715 "Pallet_prepick" "breakAfter"
    movej(get_inverse_kin(pose_trans(Pallet_prepick_p, get_tcp_offset()), qnear=Pallet_prepick_q), a=1.3962634015954636, v=1.0471975511965976)
    $ 716 "MoveL"
    $ 717 "Pick_canister" "breakAfter"
    movel(pose_trans(Pick_canister_p, get_tcp_offset()), a=1.2, v=0.25)
    $ 718 "Set OuTNET_Gripper=6"
    write_output_integer_register(0, 6)
    $ 719 "Set OutNet_Tool=On"
    write_output_boolean_register(2, True)
    $ 720 "Wait: 3.0"
    sleep(3.0)
    $ 721 "Wait InNET_InPos=HI"
    while (read_input_boolean_register(1) == False):
      sync()
    end
    $ 722 "Set OutNet_Tool=Off"
    write_output_boolean_register(2, False)
    $ 723 "MoveL"
    $ 724 "Pallet_prepick" "breakAfter"
    movel(pose_trans(Pallet_prepick_p, get_tcp_offset()), a=1.2, v=0.25)
    $ 725 "MoveJ"
    $ 726 "Canister_aprox" "breakAfter"
    movej(get_inverse_kin(Canister_aprox_p, qnear=Canister_aprox_q), a=1.3962634015954636, v=1.0471975511965976)
    $ 727 "MoveL"
    $ 728 "pl1Canister23up" "breakAfter"
    movel(pose_trans(Plane_1_Pack, pose_trans(p[.061451264231, -.289311417922, -.073379282729, -.000157706105, .000169116670, 2.356123162082], pl1Canister23up_p)), a=1.2, v=0.25)
    $ 729 "MoveL"
    $ 730 "pl1Canister23" "breakAfter"
    movel(pose_trans(Plane_1_Pack, pose_trans(p[.061451264231, -.289311417922, -.073379282729, -.000157706105, .000169116670, 2.356123162082], pl1Canister23_p)), a=1.2, v=0.25)
    $ 731 "Set OuTNET_Gripper=2"
    write_output_integer_register(0, 2)
    $ 732 "Set OutNet_Tool=On"
    write_output_boolean_register(2, True)
    $ 733 "Wait: 3.0"
    sleep(3.0)
    $ 734 "Wait InNET_InPos=HI"
    while (read_input_boolean_register(1) == False):
      sync()
    end
    $ 735 "Set OutNet_Tool=Off"
    write_output_boolean_register(2, False)
    $ 736 "MoveL"
    $ 737 "pl1Canist23up" "breakAfter"
    movel(pose_trans(Plane_1_Pack, pose_trans(p[.061451264231, -.289311417922, -.073379282729, -.000157706105, .000169116670, 2.356123162082], pl1Canist23up_p)), a=1.2, v=0.25)
    $ 738 "MoveJ"
    $ 739 "Canister_aprox" "breakAfter"
    movej(get_inverse_kin(Canister_aprox_p, qnear=Canister_aprox_q), a=1.3962634015954636, v=1.0471975511965976)
  end
  def PK2CAN4_release():
    $ 740 "PK2CAN4_release" "noBreak"
    $ 741 "MoveJ"
    $ 742 "Pallet_prepick" "breakAfter"
    movej(get_inverse_kin(pose_trans(Pallet_prepick_p, get_tcp_offset()), qnear=Pallet_prepick_q), a=1.3962634015954636, v=1.0471975511965976)
    $ 743 "MoveL"
    $ 744 "Pick_canister" "breakAfter"
    movel(pose_trans(Pick_canister_p, get_tcp_offset()), a=1.2, v=0.25)
    $ 745 "Set OuTNET_Gripper=6"
    write_output_integer_register(0, 6)
    $ 746 "Set OutNet_Tool=On"
    write_output_boolean_register(2, True)
    $ 747 "Wait: 3.0"
    sleep(3.0)
    $ 748 "Wait InNET_InPos=HI"
    while (read_input_boolean_register(1) == False):
      sync()
    end
    $ 749 "Set OutNet_Tool=Off"
    write_output_boolean_register(2, False)
    $ 750 "MoveL"
    $ 751 "Pallet_prepick" "breakAfter"
    movel(pose_trans(Pallet_prepick_p, get_tcp_offset()), a=1.2, v=0.25)
    $ 752 "MoveJ"
    $ 753 "Canister_aprox" "breakAfter"
    movej(get_inverse_kin(Canister_aprox_p, qnear=Canister_aprox_q), a=1.3962634015954636, v=1.0471975511965976)
    $ 754 "MoveL"
    $ 755 "pl1Canister24up" "breakAfter"
    movel(pose_trans(Plane_1_Pack, pose_trans(p[.061451264231, -.289311417922, -.073379282729, -.000157706105, .000169116670, 2.356123162082], pl1Canister24up_p)), a=1.2, v=0.25)
    $ 756 "MoveL"
    $ 757 "pl1Canister24" "breakAfter"
    movel(pose_trans(Plane_1_Pack, pose_trans(p[.061451264231, -.289311417922, -.073379282729, -.000157706105, .000169116670, 2.356123162082], pl1Canister24_p)), a=1.2, v=0.25)
    $ 758 "Set OuTNET_Gripper=2"
    write_output_integer_register(0, 2)
    $ 759 "Set OutNet_Tool=On"
    write_output_boolean_register(2, True)
    $ 760 "Wait: 3.0"
    sleep(3.0)
    $ 761 "Wait InNET_InPos=HI"
    while (read_input_boolean_register(1) == False):
      sync()
    end
    $ 762 "Set OutNet_Tool=Off"
    write_output_boolean_register(2, False)
    $ 763 "MoveL"
    $ 764 "pl1Canist24up" "breakAfter"
    movel(pose_trans(Plane_1_Pack, pose_trans(p[.061451264231, -.289311417922, -.073379282729, -.000157706105, .000169116670, 2.356123162082], pl1Canist24up_p)), a=1.2, v=0.25)
    $ 765 "MoveJ"
    $ 766 "Canister_aprox" "breakAfter"
    movej(get_inverse_kin(Canister_aprox_p, qnear=Canister_aprox_q), a=1.3962634015954636, v=1.0471975511965976)
  end
  def PK3CAN1_release():
    $ 767 "PK3CAN1_release" "noBreak"
    $ 768 "MoveJ"
    $ 769 "Pallet_prepick" "breakAfter"
    movej(get_inverse_kin(pose_trans(Pallet_prepick_p, get_tcp_offset()), qnear=Pallet_prepick_q), a=1.3962634015954636, v=1.0471975511965976)
    $ 770 "MoveL"
    $ 771 "Pick_canister" "breakAfter"
    movel(pose_trans(Pick_canister_p, get_tcp_offset()), a=1.2, v=0.25)
    $ 772 "Set OuTNET_Gripper=6"
    write_output_integer_register(0, 6)
    $ 773 "Set OutNet_Tool=On"
    write_output_boolean_register(2, True)
    $ 774 "Wait: 3.0"
    sleep(3.0)
    $ 775 "Wait InNET_InPos=HI"
    while (read_input_boolean_register(1) == False):
      sync()
    end
    $ 776 "Set OutNet_Tool=Off"
    write_output_boolean_register(2, False)
    $ 777 "MoveL"
    $ 778 "Pallet_prepick" "breakAfter"
    movel(pose_trans(Pallet_prepick_p, get_tcp_offset()), a=1.2, v=0.25)
    $ 779 "MoveJ"
    $ 780 "Canister_aprox" "breakAfter"
    movej(get_inverse_kin(Canister_aprox_p, qnear=Canister_aprox_q), a=1.3962634015954636, v=1.0471975511965976)
    $ 781 "MoveL"
    $ 782 "pl1Canister31up" "breakAfter"
    movel(pose_trans(Plane_1_Pack, pose_trans(p[.061451264231, -.289311417922, -.073379282729, -.000157706105, .000169116670, 2.356123162082], pl1Canister31up_p)), a=1.2, v=0.25)
    $ 783 "MoveL"
    $ 784 "pl1Canister31" "breakAfter"
    movel(pose_trans(Plane_1_Pack, pose_trans(p[.061451264231, -.289311417922, -.073379282729, -.000157706105, .000169116670, 2.356123162082], pl1Canister31_p)), a=1.2, v=0.25)
    $ 785 "Set OuTNET_Gripper=2"
    write_output_integer_register(0, 2)
    $ 786 "Set OutNet_Tool=On"
    write_output_boolean_register(2, True)
    $ 787 "Wait: 3.0"
    sleep(3.0)
    $ 788 "Wait InNET_InPos=HI"
    while (read_input_boolean_register(1) == False):
      sync()
    end
    $ 789 "Set OutNet_Tool=Off"
    write_output_boolean_register(2, False)
    $ 790 "MoveL"
    $ 791 "pl1Canist31up" "breakAfter"
    movel(pose_trans(Plane_1_Pack, pose_trans(p[.061451264231, -.289311417922, -.073379282729, -.000157706105, .000169116670, 2.356123162082], pl1Canist31up_p)), a=1.2, v=0.25)
    $ 792 "MoveJ"
    $ 793 "Canister_aprox" "breakAfter"
    movej(get_inverse_kin(Canister_aprox_p, qnear=Canister_aprox_q), a=1.3962634015954636, v=1.0471975511965976)
  end
  def PK3CAN2_release():
    $ 794 "PK3CAN2_release" "noBreak"
    $ 795 "MoveJ"
    $ 796 "Pallet_prepick" "breakAfter"
    movej(get_inverse_kin(pose_trans(Pallet_prepick_p, get_tcp_offset()), qnear=Pallet_prepick_q), a=1.3962634015954636, v=1.0471975511965976)
    $ 797 "MoveL"
    $ 798 "Pick_canister" "breakAfter"
    movel(pose_trans(Pick_canister_p, get_tcp_offset()), a=1.2, v=0.25)
    $ 799 "Set OuTNET_Gripper=6"
    write_output_integer_register(0, 6)
    $ 800 "Set OutNet_Tool=On"
    write_output_boolean_register(2, True)
    $ 801 "Wait: 3.0"
    sleep(3.0)
    $ 802 "Wait InNET_InPos=HI"
    while (read_input_boolean_register(1) == False):
      sync()
    end
    $ 803 "Set OutNet_Tool=Off"
    write_output_boolean_register(2, False)
    $ 804 "MoveL"
    $ 805 "Pallet_prepick" "breakAfter"
    movel(pose_trans(Pallet_prepick_p, get_tcp_offset()), a=1.2, v=0.25)
    $ 806 "MoveJ"
    $ 807 "Canister_aprox" "breakAfter"
    movej(get_inverse_kin(Canister_aprox_p, qnear=Canister_aprox_q), a=1.3962634015954636, v=1.0471975511965976)
    $ 808 "MoveL"
    $ 809 "pl1Canister32up" "breakAfter"
    movel(pose_trans(Plane_1_Pack, pose_trans(p[.061451264231, -.289311417922, -.073379282729, -.000157706105, .000169116670, 2.356123162082], pl1Canister32up_p)), a=1.2, v=0.25)
    $ 810 "MoveL"
    $ 811 "pl1Canister32" "breakAfter"
    movel(pose_trans(Plane_1_Pack, pose_trans(p[.061451264231, -.289311417922, -.073379282729, -.000157706105, .000169116670, 2.356123162082], pl1Canister32_p)), a=1.2, v=0.25)
    $ 812 "Set OuTNET_Gripper=2"
    write_output_integer_register(0, 2)
    $ 813 "Set OutNet_Tool=On"
    write_output_boolean_register(2, True)
    $ 814 "Wait: 3.0"
    sleep(3.0)
    $ 815 "Wait InNET_InPos=HI"
    while (read_input_boolean_register(1) == False):
      sync()
    end
    $ 816 "Set OutNet_Tool=Off"
    write_output_boolean_register(2, False)
    $ 817 "MoveL"
    $ 818 "pl1Canist32up" "breakAfter"
    movel(pose_trans(Plane_1_Pack, pose_trans(p[.061451264231, -.289311417922, -.073379282729, -.000157706105, .000169116670, 2.356123162082], pl1Canist32up_p)), a=1.2, v=0.25)
    $ 819 "MoveJ"
    $ 820 "Canister_aprox" "breakAfter"
    movej(get_inverse_kin(Canister_aprox_p, qnear=Canister_aprox_q), a=1.3962634015954636, v=1.0471975511965976)
  end
  def PK3CAN3_release():
    $ 821 "PK3CAN3_release" "noBreak"
    $ 822 "MoveJ"
    $ 823 "Pallet_prepick" "breakAfter"
    movej(get_inverse_kin(pose_trans(Pallet_prepick_p, get_tcp_offset()), qnear=Pallet_prepick_q), a=1.3962634015954636, v=1.0471975511965976)
    $ 824 "MoveL"
    $ 825 "Pick_canister" "breakAfter"
    movel(pose_trans(Pick_canister_p, get_tcp_offset()), a=1.2, v=0.25)
    $ 826 "Set OuTNET_Gripper=6"
    write_output_integer_register(0, 6)
    $ 827 "Set OutNet_Tool=On"
    write_output_boolean_register(2, True)
    $ 828 "Wait: 3.0"
    sleep(3.0)
    $ 829 "Wait InNET_InPos=HI"
    while (read_input_boolean_register(1) == False):
      sync()
    end
    $ 830 "Set OutNet_Tool=Off"
    write_output_boolean_register(2, False)
    $ 831 "MoveL"
    $ 832 "Pallet_prepick" "breakAfter"
    movel(pose_trans(Pallet_prepick_p, get_tcp_offset()), a=1.2, v=0.25)
    $ 833 "MoveJ"
    $ 834 "Canister_aprox" "breakAfter"
    movej(get_inverse_kin(Canister_aprox_p, qnear=Canister_aprox_q), a=1.3962634015954636, v=1.0471975511965976)
    $ 835 "MoveL"
    $ 836 "pl1Canister33up" "breakAfter"
    movel(pose_trans(Plane_1_Pack, pose_trans(p[.061451264231, -.289311417922, -.073379282729, -.000157706105, .000169116670, 2.356123162082], pl1Canister33up_p)), a=1.2, v=0.25)
    $ 837 "MoveL"
    $ 838 "pl1Canister33" "breakAfter"
    movel(pose_trans(Plane_1_Pack, pose_trans(p[.061451264231, -.289311417922, -.073379282729, -.000157706105, .000169116670, 2.356123162082], pl1Canister33_p)), a=1.2, v=0.25)
    $ 839 "Set OuTNET_Gripper=2"
    write_output_integer_register(0, 2)
    $ 840 "Set OutNet_Tool=On"
    write_output_boolean_register(2, True)
    $ 841 "Wait: 3.0"
    sleep(3.0)
    $ 842 "Wait InNET_InPos=HI"
    while (read_input_boolean_register(1) == False):
      sync()
    end
    $ 843 "Set OutNet_Tool=Off"
    write_output_boolean_register(2, False)
    $ 844 "MoveL"
    $ 845 "pl1Canist3up" "breakAfter"
    movel(pose_trans(Plane_1_Pack, pose_trans(p[.061451264231, -.289311417922, -.073379282729, -.000157706105, .000169116670, 2.356123162082], pl1Canist3up_p)), a=1.2, v=0.25)
    $ 846 "MoveJ"
    $ 847 "Canister_aprox" "breakAfter"
    movej(get_inverse_kin(Canister_aprox_p, qnear=Canister_aprox_q), a=1.3962634015954636, v=1.0471975511965976)
  end
  def PK3CAN4_release():
    $ 848 "PK3CAN4_release" "noBreak"
    $ 849 "MoveJ"
    $ 850 "Pallet_prepick" "breakAfter"
